	X =  247.902  mm,	Y =   -382.009  mm,	Z =   -256.245  mm,
	W =  90.000 deg,	P =   0.000 deg,	R =   90.000 deg
};
P[319]{
   GP1:
	UF : 0, UT : 6,		CONFIG : 'N U T, 0, 0, 0',
	X =  248.616  mm,	Y =   -381.594  mm,	Z =   -256.279  mm,
	W =  90.000 deg,	P =   0.000 deg,	R =   90.000 deg
};
P[320]{
   GP1:
	UF : 0, UT : 6,		CONFIG : 'N U T, 0, 0, 0',
	X =  254.561  mm,	Y =   -378.161  mm,	Z =   -256.286  mm,
	W =  90.000 deg,	P =   0.000 deg,	R =   90.000 deg
};
P[321]{
   GP1:
	UF : 0, UT : 6,		CONFIG : 'N U T, 0, 0, 0',
	X =  255.267  mm,	Y =   -377.759  mm,	Z =   -256.214  mm,
	W =  90.000 deg,	P =   0.000 deg,	R =   90.000 deg
};
P[322]{
   GP1:
	UF : 0, UT : 6,		CONFIG : 'N U T, 0, 0, 0',
	X =  258.215  mm,	Y =   -376.051  mm,	Z =   -256.285  mm,
	W =  90.000 deg,	P =   0.000 deg,	R =   90.000 deg
};
P[323]{
   GP1:
	UF : 0, UT : 6,		CONFIG : 'N U T, 0, 0, 0',
	X =  261.977  mm,	Y =   -373.884  mm,	Z =   -256.215  mm,
	W =  90.000 deg,	P =   0.000 deg,	R =   90.000 deg
};
P[324]{
   GP1:
	UF : 0, UT : 6,		CONFIG : 'N U T, 0, 0, 0',
	X =  262.661  mm,	Y =   -373.497  mm,	Z =   -256.123  mm,
	W =  90.000 deg,	P =   0.000 deg,	R =   90.000 deg
};
P[325]{
   GP1:
	UF : 0, UT : 6,		CONFIG : 'N U T, 0, 0, 0',
	X =  263.369  mm,	Y =   -373.079  mm,	Z =   -256.244  mm,
	W =  90.000 deg,	P =   0.000 deg,	R =   90.000 deg
};
P[326]{
   GP1:
	UF : 0, UT : 6,		CONFIG : 'N U T, 0, 0, 0',
	X =  265.622  mm,	Y =   -371.779  mm,	Z =   -256.224  mm,
	W =  90.000 deg,	P =   0.000 deg,	R =   90.000 deg
};
P[327]{
   GP1:
	UF : 0, UT : 6,		CONFIG : 'N U T, 0, 0, 0',
	X =  267.023  mm,	Y =   -370.977  mm,	Z =   -256.135  mm,
	W =  90.000 deg,	P =   0.000 deg,	R =   90.000 deg
};
P[328]{
   GP1:
	UF : 0, UT : 6,		CONFIG : 'N U T, 0, 0, 0',
	X =  267.777  mm,	Y =   -370.522  mm,	Z =   -256.283  mm,
	W =  90.000 deg,	P =   0.000 deg,	R =   90.000 deg
};
P[329]{
   GP1:
	UF : 0, UT : 6,		CONFIG : 'N U T, 0, 0, 0',
	X =  269.721  mm,	Y =   -369.001  mm,	Z =   -256.087  mm,
	W =  90.000 deg,	P =   0.000 deg,	R =   90.000 deg
};
P[330]{
   GP1:
	UF : 0, UT : 6,		CONFIG : 'N U T, 0, 0, 0',
	X =  269.875  mm,	Y =   -368.853  mm,	Z =   -255.819  mm,
	W =  90.000 deg,	P =   0.000 deg,	R =   90.000 deg
};
P[331]{
   GP1:
	UF : 0, UT : 6,		CONFIG : 'N U T, 0, 0, 0',
	X =  270.416  mm,	Y =   -368.129  mm,	Z =   -256.212  mm,
	W =  90.000 deg,	P =   0.000 deg,	R =   90.000 deg
};
P[332]{
   GP1:
	UF : 0, UT : 6,		CONFIG : 'N U T, 0, 0, 0',
	X =  270.805  mm,	Y =   -367.534  mm,	Z =   -256.111  mm,
	W =  90.000 deg,	P =   0.000 deg,	R =   90.000 deg
};
P[333]{
   GP1:
	UF : 0, UT : 6,		CONFIG : 'N U T, 0, 0, 0',
	X =  270.994  mm,	Y =   -367.194  mm,	Z =   -256.250  mm,
	W =  90.000 deg,	P =   0.000 deg,	R =   90.000 deg
};
P[334]{
   GP1:
	UF : 0, UT : 6,		CONFIG : 'N U T, 0, 0, 0',
	X =  271.729  mm,	Y =   -365.277  mm,	Z =   -256.239  mm,
	W =  90.000 deg,	P =   0.000 deg,	R =   90.000 deg
};
P[335]{
   GP1:
	UF : 0, UT : 6,		CONFIG : 'N U T, 0, 0, 0',
	X =  271.851  mm,	Y =   -361.616  mm,	Z =   -256.115  mm,
	W =  90.000 deg,	P =   0.000 deg,	R =   90.000 deg
};
P[336]{
   GP1:
	UF : 0, UT : 6,		CONFIG : 'N U T, 0, 0, 0',
	X =  271.727  mm,	Y =   -361.053  mm,	Z =   -256.193  mm,
	W =  90.000 deg,	P =   0.000 deg,	R =   90.000 deg
};
P[337]{
   GP1:
	UF : 0, UT : 6,		CONFIG : 'N U T, 0, 0, 0',
	X =  270.444  mm,	Y =   -358.219  mm,	Z =   -256.266  mm,
	W =  90.000 deg,	P =   0.000 deg,	R =   90.000 deg
};
P[338]{
   GP1:
	UF : 0, UT : 6,		CONFIG : 'N U T, 0, 0, 0',
	X =  270.041  mm,	Y =   -357.511  mm,	Z =   -256.196  mm,
	W =  90.000 deg,	P =   0.000 deg,	R =   90.000 deg
};
P[339]{
   GP1:
	UF : 0, UT : 6,		CONFIG : 'N U T, 0, 0, 0',
	X =  268.750  mm,	Y =   -355.278  mm,	Z =   -256.223  mm,
	W =  90.000 deg,	P =   0.000 deg,	R =   90.000 deg
};
P[340]{
   GP1:
	UF : 0, UT : 6,		CONFIG : 'N U T, 0, 0, 0',
	X =  267.926  mm,	Y =   -353.854  mm,	Z =   -256.236  mm,
	W =  90.000 deg,	P =   0.000 deg,	R =   90.000 deg
};
P[341]{
   GP1:
	UF : 0, UT : 6,		CONFIG : 'N U T, 0, 0, 0',
	X =  266.617  mm,	Y =   -351.583  mm,	Z =   -256.210  mm,
	W =  90.000 deg,	P =   0.000 deg,	R =   90.000 deg
};
P[342]{
   GP1:
	UF : 0, UT : 6,		CONFIG : 'N U T, 0, 0, 0',
	X =  265.790  mm,	Y =   -350.160  mm,	Z =   -256.269  mm,
	W =  90.000 deg,	P =   0.000 deg,	R =   90.000 deg
};
P[343]{
   GP1:
	UF : 0, UT : 6,		CONFIG : 'N U T, 0, 0, 0',
	X =  265.369  mm,	Y =   -349.416  mm,	Z =   -256.174  mm,
	W =  90.000 deg,	P =   0.000 deg,	R =   90.000 deg
};
P[344]{
   GP1:
	UF : 0, UT : 6,		CONFIG : 'N U T, 0, 0, 0',
	X =  264.933  mm,	Y =   -348.670  mm,	Z =   -256.231  mm,
	W =  90.000 deg,	P =   0.000 deg,	R =   90.000 deg
};
P[345]{
   GP1:
	UF : 0, UT : 6,		CONFIG : 'N U T, 0, 0, 0',
	X =  264.491  mm,	Y =   -347.910  mm,	Z =   -256.272  mm,
	W =  90.000 deg,	P =   0.000 deg,	R =   90.000 deg
};
P[346]{
   GP1:
	UF : 0, UT : 6,		CONFIG : 'N U T, 0, 0, 0',
	X =  264.090  mm,	Y =   -347.215  mm,	Z =   -256.262  mm,
	W =  90.000 deg,	P =   0.000 deg,	R =   90.000 deg
};
P[347]{
   GP1:
	UF : 0, UT : 6,		CONFIG : 'N U T, 0, 0, 0',
	X =  262.830  mm,	Y =   -345.031  mm,	Z =   -256.263  mm,
	W =  90.000 deg,	P =   0.000 deg,	R =   90.000 deg
};
P[348]{
   GP1:
	UF : 0, UT : 6,		CONFIG : 'N U T, 0, 0, 0',
	X =  262.368  mm,	Y =   -344.233  mm,	Z =   -256.279  mm,
	W =  90.000 deg,	P =   0.000 deg,	R =   90.000 deg
};
P[349]{
   GP1:
	UF : 0, UT : 6,		CONFIG : 'N U T, 0, 0, 0',
	X =  262.026  mm,	Y =   -343.628  mm,	Z =   -256.184  mm,
	W =  90.000 deg,	P =   0.000 deg,	R =   90.000 deg
};
P[350]{
   GP1:
	UF : 0, UT : 6,		CONFIG : 'N U T, 0, 0, 0',
	X =  260.236  mm,	Y =   -340.533  mm,	Z =   -256.219  mm,
	W =  90.000 deg,	P =   0.000 deg,	R =   90.000 deg
};
P[351]{
   GP1:
	UF : 0, UT : 6,		CONFIG : 'N U T, 0, 0, 0',
	X =  259.438  mm,	Y =   -339.161  mm,	Z =   -256.290  mm,
	W =  90.000 deg,	P =   0.000 deg,	R =   90.000 deg
};
P[352]{
   GP1:
	UF : 0, UT : 6,		CONFIG : 'N U T, 0, 0, 0',
	X =  258.110  mm,	Y =   -336.856  mm,	Z =   -256.255  mm,
	W =  90.000 deg,	P =   0.000 deg,	R =   90.000 deg
};
P[353]{
   GP1:
	UF : 0, UT : 6,		CONFIG : 'N U T, 0, 0, 0',
	X =  257.689  mm,	Y =   -336.131  mm,	Z =   -256.291  mm,
	W =  90.000 deg,	P =   0.000 deg,	R =   90.000 deg
};
P[354]{
   GP1:
	UF : 0, UT : 6,		CONFIG : 'N U T, 0, 0, 0',
	X =  256.431  mm,	Y =   -333.937  mm,	Z =   -256.170  mm,
	W =  90.000 deg,	P =   0.000 deg,	R =   90.000 deg
};
P[355]{
   GP1:
	UF : 0, UT : 6,		CONFIG : 'N U T, 0, 0, 0',
	X =  255.567  mm,	Y =   -332.445  mm,	Z =   -256.199  mm,
	W =  90.000 deg,	P =   0.000 deg,	R =   90.000 deg
};
P[356]{
   GP1:
	UF : 0, UT : 6,		CONFIG : 'N U T, 0, 0, 0',
	X =  255.156  mm,	Y =   -331.729  mm,	Z =   -256.181  mm,
	W =  90.000 deg,	P =   0.000 deg,	R =   90.000 deg
};
P[357]{
   GP1:
	UF : 0, UT : 6,		CONFIG : 'N U T, 0, 0, 0',
	X =  254.665  mm,	Y =   -330.894  mm,	Z =   -256.283  mm,
	W =  90.000 deg,	P =   0.000 deg,	R =   90.000 deg
};
P[358]{
   GP1:
	UF : 0, UT : 6,		CONFIG : 'N U T, 0, 0, 0',
	X =  254.295  mm,	Y =   -330.269  mm,	Z =   -256.272  mm,
	W =  90.000 deg,	P =   0.000 deg,	R =   90.000 deg
};
P[359]{
   GP1:
	UF : 0, UT : 6,		CONFIG : 'N U T, 0, 0, 0',
	X =  253.269  mm,	Y =   -328.882  mm,	Z =   -256.236  mm,
	W =  90.000 deg,	P =   0.000 deg,	R =   90.000 deg
};
P[360]{
   GP1:
	UF : 0, UT : 6,		CONFIG : 'N U T, 0, 0, 0',
	X =  252.851  mm,	Y =   -328.417  mm,	Z =   -256.192  mm,
	W =  90.000 deg,	P =   0.000 deg,	R =   90.000 deg
};
P[361]{
   GP1:
	UF : 0, UT : 6,		CONFIG : 'N U T, 0, 0, 0',
	X =  252.558  mm,	Y =   -328.182  mm,	Z =   -256.287  mm,
	W =  90.000 deg,	P =   0.000 deg,	R =   90.000 deg
};
P[362]{
   GP1:
	UF : 0, UT : 6,		CONFIG : 'N U T, 0, 0, 0',
	X =  251.892  mm,	Y =   -327.641  mm,	Z =   -256.229  mm,
	W =  90.000 deg,	P =   0.000 deg,	R =   90.000 deg
};
P[363]{
   GP1:
	UF : 0, UT : 6,		CONFIG : 'N U T, 0, 0, 0',
	X =  251.459  mm,	Y =   -327.358  mm,	Z =   -256.187  mm,
	W =  90.000 deg,	P =   0.000 deg,	R =   90.000 deg
};
P[364]{
   GP1:
	UF : 0, UT : 6,		CONFIG : 'N U T, 0, 0, 0',
	X =  249.222  mm,	Y =   -326.377  mm,	Z =   -256.167  mm,
	W =  90.000 deg,	P =   0.000 deg,	R =   90.000 deg
};
P[365]{
   GP1:
	UF : 0, UT : 6,		CONFIG : 'N U T, 0, 0, 0',
	X =  248.144  mm,	Y =   -326.165  mm,	Z =   -256.273  mm,
	W =  90.000 deg,	P =   0.000 deg,	R =   90.000 deg
};
P[366]{
   GP1:
	UF : 0, UT : 6,		CONFIG : 'N U T, 0, 0, 0',
	X =  247.391  mm,	Y =   -326.065  mm,	Z =   -256.154  mm,
	W =  90.000 deg,	P =   0.000 deg,	R =   90.000 deg
};
P[367]{
   GP1:
	UF : 0, UT : 6,		CONFIG : 'N U T, 0, 0, 0',
	X =  246.118  mm,	Y =   -326.120  mm,	Z =   -256.195  mm,
	W =  90.000 deg,	P =   0.000 deg,	R =   90.000 deg
};
P[368]{
   GP1:
	UF : 0, UT : 6,		CONFIG : 'N U T, 0, 0, 0',
	X =  244.973  mm,	Y =   -326.275  mm,	Z =   -255.877  mm,
	W =  90.000 deg,	P =   0.000 deg,	R =   90.000 deg
};
P[369]{
   GP1:
	UF : 0, UT : 6,		CONFIG : 'N U T, 0, 0, 0',
	X =  244.461  mm,	Y =   -326.465  mm,	Z =   -256.182  mm,
	W =  90.000 deg,	P =   0.000 deg,	R =   90.000 deg
};
P[370]{
   GP1:
	UF : 0, UT : 6,		CONFIG : 'N U T, 0, 0, 0',
	X =  242.026  mm,	Y =   -327.612  mm,	Z =   -256.201  mm,
	W =  90.000 deg,	P =   0.000 deg,	R =   90.000 deg
};
P[371]{
   GP1:
	UF : 0, UT : 6,		CONFIG : 'N U T, 0, 0, 0',
	X =  241.272  mm,	Y =   -328.043  mm,	Z =   -256.156  mm,
	W =  90.000 deg,	P =   0.000 deg,	R =   90.000 deg
};
P[372]{
   GP1:
	UF : 0, UT : 6,		CONFIG : 'N U T, 0, 0, 0',
	X =  240.597  mm,	Y =   -328.438  mm,	Z =   -256.220  mm,
	W =  90.000 deg,	P =   0.000 deg,	R =   90.000 deg
};
P[373]{
   GP1:
	UF : 0, UT : 6,		CONFIG : 'N U T, 0, 0, 0',
	X =  239.869  mm,	Y =   -328.863  mm,	Z =   -256.275  mm,
	W =  90.000 deg,	P =   0.000 deg,	R =   90.000 deg
};
P[374]{
   GP1:
	UF : 0, UT : 6,		CONFIG : 'N U T, 0, 0, 0',
	X =  239.046  mm,	Y =   -329.332  mm,	Z =   -256.198  mm,
	W =  90.000 deg,	P =   0.000 deg,	R =   90.000 deg
};
P[375]{
   GP1:
	UF : 0, UT : 6,		CONFIG : 'N U T, 0, 0, 0',
	X =  236.149  mm,	Y =   -331.005  mm,	Z =   -256.201  mm,
	W =  90.000 deg,	P =   0.000 deg,	R =   90.000 deg
};
P[376]{
   GP1:
	UF : 0, UT : 6,		CONFIG : 'N U T, 0, 0, 0',
	X =  234.723  mm,	Y =   -331.834  mm,	Z =   -256.270  mm,
	W =  90.000 deg,	P =   0.000 deg,	R =   90.000 deg
};
P[377]{
   GP1:
	UF : 0, UT : 6,		CONFIG : 'N U T, 0, 0, 0',
	X =  233.937  mm,	Y =   -332.289  mm,	Z =   -256.289  mm,
	W =  90.000 deg,	P =   0.000 deg,	R =   90.000 deg
};
P[378]{
   GP1:
	UF : 0, UT : 6,		CONFIG : 'N U T, 0, 0, 0',
	X =  233.257  mm,	Y =   -332.681  mm,	Z =   -256.279  mm,
	W =  90.000 deg,	P =   0.000 deg,	R =   90.000 deg
};
P[379]{
   GP1:
	UF : 0, UT : 6,		CONFIG : 'N U T, 0, 0, 0',
	X =  232.524  mm,	Y =   -333.105  mm,	Z =   -256.284  mm,
	W =  90.000 deg,	P =   0.000 deg,	R =   90.000 deg
};
P[380]{
   GP1:
	UF : 0, UT : 6,		CONFIG : 'N U T, 0, 0, 0',
	X =  231.761  mm,	Y =   -333.543  mm,	Z =   -256.260  mm,
	W =  90.000 deg,	P =   0.000 deg,	R =   90.000 deg
};
P[381]{
   GP1:
	UF : 0, UT : 6,		CONFIG : 'N U T, 0, 0, 0',
	X =  230.964  mm,	Y =   -333.998  mm,	Z =   -256.198  mm,
	W =  90.000 deg,	P =   0.000 deg,	R =   90.000 deg
};
P[382]{
   GP1:
	UF : 0, UT : 6,		CONFIG : 'N U T, 0, 0, 0',
	X =  230.308  mm,	Y =   -334.378  mm,	Z =   -256.209  mm,
	W =  90.000 deg,	P =   0.000 deg,	R =   90.000 deg
};
P[383]{
   GP1:
	UF : 0, UT : 6,		CONFIG : 'N U T, 0, 0, 0',
	X =  228.762  mm,	Y =   -335.273  mm,	Z =   -256.235  mm,
	W =  90.000 deg,	P =   0.000 deg,	R =   90.000 deg
};
P[384]{
   GP1:
	UF : 0, UT : 6,		CONFIG : 'N U T, 0, 0, 0',
	X =  226.535  mm,	Y =   -336.563  mm,	Z =   -256.285  mm,
	W =  90.000 deg,	P =   0.000 deg,	R =   90.000 deg
};
P[385]{
   GP1:
	UF : 0, UT : 6,		CONFIG : 'N U T, 0, 0, 0',
	X =  225.039  mm,	Y =   -337.426  mm,	Z =   -256.282  mm,
	W =  90.000 deg,	P =   0.000 deg,	R =   90.000 deg
};
P[386]{
   GP1:
	UF : 0, UT : 6,		CONFIG : 'N U T, 0, 0, 0',
	X =  224.460  mm,	Y =   -337.761  mm,	Z =   -256.294  mm,
	W =  90.000 deg,	P =   0.000 deg,	R =   90.000 deg
};
P[387]{
   GP1:
	UF : 0, UT : 6,		CONFIG : 'N U T, 0, 0, 0',
	X =  222.903  mm,	Y =   -338.653  mm,	Z =   -256.193  mm,
	W =  90.000 deg,	P =   0.000 deg,	R =   90.000 deg
};
P[388]{
   GP1:
	UF : 0, UT : 6,		CONFIG : 'N U T, 0, 0, 0',
	X =  218.417  mm,	Y =   -341.244  mm,	Z =   -256.213  mm,
	W =  90.000 deg,	P =   0.000 deg,	R =   90.000 deg
};
P[389]{
   GP1:
	UF : 0, UT : 6,		CONFIG : 'N U T, 0, 0, 0',
	X =  217.647  mm,	Y =   -341.694  mm,	Z =   -256.278  mm,
	W =  90.000 deg,	P =   0.000 deg,	R =   90.000 deg
};
P[390]{
   GP1:
	UF : 0, UT : 6,		CONFIG : 'N U T, 0, 0, 0',
	X =  214.021  mm,	Y =   -343.783  mm,	Z =   -256.220  mm,
	W =  90.000 deg,	P =   0.000 deg,	R =   90.000 deg
};
P[391]{
   GP1:
	UF : 0, UT : 6,		CONFIG : 'N U T, 0, 0, 0',
	X =  212.512  mm,	Y =   -344.659  mm,	Z =   -256.271  mm,
	W =  90.000 deg,	P =   0.000 deg,	R =   90.000 deg
};
P[392]{
   GP1:
	UF : 0, UT : 6,		CONFIG : 'N U T, 0, 0, 0',
	X =  211.156  mm,	Y =   -345.440  mm,	Z =   -256.255  mm,
	W =  90.000 deg,	P =   0.000 deg,	R =   90.000 deg
};
P[393]{
   GP1:
	UF : 0, UT : 6,		CONFIG : 'N U T, 0, 0, 0',
	X =  210.447  mm,	Y =   -345.848  mm,	Z =   -256.237  mm,
	W =  90.000 deg,	P =   0.000 deg,	R =   90.000 deg
};
P[394]{
   GP1:
	UF : 0, UT : 6,		CONFIG : 'N U T, 0, 0, 0',
	X =  208.242  mm,	Y =   -347.121  mm,	Z =   -256.243  mm,
	W =  90.000 deg,	P =   0.000 deg,	R =   90.000 deg
};
P[395]{
   GP1:
	UF : 0, UT : 6,		CONFIG : 'N U T, 0, 0, 0',
	X =  207.402  mm,	Y =   -347.608  mm,	Z =   -256.253  mm,
	W =  90.000 deg,	P =   0.000 deg,	R =   90.000 deg
};
P[396]{
   GP1:
	UF : 0, UT : 6,		CONFIG : 'N U T, 0, 0, 0',
	X =  205.941  mm,	Y =   -348.452  mm,	Z =   -256.265  mm,
	W =  90.000 deg,	P =   0.000 deg,	R =   90.000 deg
};
P[397]{
   GP1:
	UF : 0, UT : 6,		CONFIG : 'N U T, 0, 0, 0',
	X =  205.190  mm,	Y =   -348.882  mm,	Z =   -256.221  mm,
	W =  90.000 deg,	P =   0.000 deg,	R =   90.000 deg
};
P[398]{
   GP1:
	UF : 0, UT : 6,		CONFIG : 'N U T, 0, 0, 0',
	X =  202.336  mm,	Y =   -350.530  mm,	Z =   -256.224  mm,
	W =  90.000 deg,	P =   0.000 deg,	R =   90.000 deg
};
P[399]{
   GP1:
	UF : 0, UT : 6,		CONFIG : 'N U T, 0, 0, 0',
	X =  200.125  mm,	Y =   -351.810  mm,	Z =   -256.270  mm,
	W =  90.000 deg,	P =   0.000 deg,	R =   90.000 deg
};
P[400]{
   GP1:
	UF : 0, UT : 6,		CONFIG : 'N U T, 0, 0, 0',
	X =  198.501  mm,	Y =   -352.750  mm,	Z =   -256.289  mm,
	W =  90.000 deg,	P =   0.000 deg,	R =   90.000 deg
};
P[401]{
   GP1:
	UF : 0, UT : 6,		CONFIG : 'N U T, 0, 0, 0',
	X =  197.783  mm,	Y =   -353.163  mm,	Z =   -256.274  mm,
	W =  90.000 deg,	P =   0.000 deg,	R =   90.000 deg
};
P[402]{
   GP1:
	UF : 0, UT : 6,		CONFIG : 'N U T, 0, 0, 0',
	X =  196.032  mm,	Y =   -353.414  mm,	Z =   -246.859  mm,
	W =  90.000 deg,	P =   0.000 deg,	R =   90.000 deg
};
P[403]{
   GP1:
	UF : 0, UT : 6,		CONFIG : 'N U T, 0, 0, 0',
	X =  195.473  mm,	Y =   -353.741  mm,	Z =   -246.915  mm,
	W =  90.000 deg,	P =   0.000 deg,	R =   90.000 deg
};
P[404]{
   GP1:
	UF : 0, UT : 6,		CONFIG : 'N U T, 0, 0, 0',
	X =  194.619  mm,	Y =   -354.233  mm,	Z =   -246.902  mm,
	W =  90.000 deg,	P =   0.000 deg,	R =   90.000 deg
};
P[405]{
   GP1:
	UF : 0, UT : 6,		CONFIG : 'N U T, 0, 0, 0',
	X =  193.731  mm,	Y =   -354.745  mm,	Z =   -246.888  mm,
	W =  90.000 deg,	P =   0.000 deg,	R =   90.000 deg
};
P[406]{
   GP1:
	UF : 0, UT : 6,		CONFIG : 'N U T, 0, 0, 0',
	X =  193.023  mm,	Y =   -355.154  mm,	Z =   -246.887  mm,
	W =  90.000 deg,	P =   0.000 deg,	R =   90.000 deg
};
P[407]{
   GP1:
	UF : 0, UT : 6,		CONFIG : 'N U T, 0, 0, 0',
	X =  192.356  mm,	Y =   -355.536  mm,	Z =   -246.860  mm,
	W =  90.000 deg,	P =   0.000 deg,	R =   90.000 deg
};
P[408]{
   GP1:
	UF : 0, UT : 6,		CONFIG : 'N U T, 0, 0, 0',
	X =  190.808  mm,	Y =   -356.432  mm,	Z =   -246.883  mm,
	W =  90.000 deg,	P =   0.000 deg,	R =   90.000 deg
};
P[409]{
   GP1:
	UF : 0, UT : 6,		CONFIG : 'N U T, 0, 0, 0',
	X =  190.217  mm,	Y =   -356.774  mm,	Z =   -246.892  mm,
	W =  90.000 deg,	P =   0.000 deg,	R =   90.000 deg
};
P[410]{
   GP1:
	UF : 0, UT : 6,		CONFIG : 'N U T, 0, 0, 0',
	X =  189.373  mm,	Y =   -357.263  mm,	Z =   -246.919  mm,
	W =  90.000 deg,	P =   0.000 deg,	R =   90.000 deg
};
P[411]{
   GP1:
	UF : 0, UT : 6,		CONFIG : 'N U T, 0, 0, 0',
	X =  188.668  mm,	Y =   -357.657  mm,	Z =   -246.758  mm,
	W =  90.000 deg,	P =   0.000 deg,	R =   90.000 deg
};
P[412]{
   GP1:
	UF : 0, UT : 6,		CONFIG : 'N U T, 0, 0, 0',
	X =  188.044  mm,	Y =   -358.028  mm,	Z =   -246.877  mm,
	W =  90.000 deg,	P =   0.000 deg,	R =   90.000 deg
};
P[413]{
   GP1:
	UF : 0, UT : 6,		CONFIG : 'N U T, 0, 0, 0',
	X =  187.147  mm,	Y =   -358.547  mm,	Z =   -246.893  mm,
	W =  90.000 deg,	P =   0.000 deg,	R =   90.000 deg
};
P[414]{
   GP1:
	UF : 0, UT : 6,		CONFIG : 'N U T, 0, 0, 0',
	X =  186.476  mm,	Y =   -358.932  mm,	Z =   -246.874  mm,
	W =  90.000 deg,	P =   0.000 deg,	R =   90.000 deg
};
P[415]{
   GP1:
	UF : 0, UT : 6,		CONFIG : 'N U T, 0, 0, 0',
	X =  185.037  mm,	Y =   -359.767  mm,	Z =   -246.923  mm,
	W =  90.000 deg,	P =   0.000 deg,	R =   90.000 deg
};
P[416]{
   GP1:
	UF : 0, UT : 6,		CONFIG : 'N U T, 0, 0, 0',
	X =  183.547  mm,	Y =   -360.627  mm,	Z =   -246.906  mm,
	W =  90.000 deg,	P =   0.000 deg,	R =   90.000 deg
};
P[417]{
   GP1:
	UF : 0, UT : 6,		CONFIG : 'N U T, 0, 0, 0',
	X =  182.141  mm,	Y =   -361.440  mm,	Z =   -246.921  mm,
	W =  90.000 deg,	P =   0.000 deg,	R =   90.000 deg
};
P[418]{
   GP1:
	UF : 0, UT : 6,		CONFIG : 'N U T, 0, 0, 0',
	X =  180.536  mm,	Y =   -362.357  mm,	Z =   -246.812  mm,
	W =  90.000 deg,	P =   0.000 deg,	R =   90.000 deg
};
P[419]{
   GP1:
	UF : 0, UT : 6,		CONFIG : 'N U T, 0, 0, 0',
	X =  178.442  mm,	Y =   -363.573  mm,	Z =   -246.894  mm,
	W =  90.000 deg,	P =   0.000 deg,	R =   90.000 deg
};
P[420]{
   GP1:
	UF : 0, UT : 6,		CONFIG : 'N U T, 0, 0, 0',
	X =  175.338  mm,	Y =   -365.357  mm,	Z =   -246.788  mm,
	W =  90.000 deg,	P =   0.000 deg,	R =   90.000 deg
};
P[421]{
   GP1:
	UF : 0, UT : 6,		CONFIG : 'N U T, 0, 0, 0',
	X =  174.572  mm,	Y =   -365.805  mm,	Z =   -246.864  mm,
	W =  90.000 deg,	P =   0.000 deg,	R =   90.000 deg
};
P[422]{
   GP1:
	UF : 0, UT : 6,		CONFIG : 'N U T, 0, 0, 0',
	X =  173.813  mm,	Y =   -366.240  mm,	Z =   -246.828  mm,
	W =  90.000 deg,	P =   0.000 deg,	R =   90.000 deg
};
P[423]{
   GP1:
	UF : 0, UT : 6,		CONFIG : 'N U T, 0, 0, 0',
	X =  173.280  mm,	Y =   -366.554  mm,	Z =   -246.906  mm,
	W =  90.000 deg,	P =   0.000 deg,	R =   90.000 deg
};
P[424]{
   GP1:
	UF : 0, UT : 6,		CONFIG : 'N U T, 0, 0, 0',
	X =  172.494  mm,	Y =   -367.005  mm,	Z =   -246.867  mm,
	W =  90.000 deg,	P =   0.000 deg,	R =   90.000 deg
};
P[425]{
   GP1:
	UF : 0, UT : 6,		CONFIG : 'N U T, 0, 0, 0',
	X =  171.741  mm,	Y =   -367.438  mm,	Z =   -246.840  mm,
	W =  90.000 deg,	P =   0.000 deg,	R =   90.000 deg
};
P[426]{
   GP1:
	UF : 0, UT : 6,		CONFIG : 'N U T, 0, 0, 0',
	X =  165.137  mm,	Y =   -371.244  mm,	Z =   -246.757  mm,
	W =  90.000 deg,	P =   0.000 deg,	R =   90.000 deg
};
P[427]{
   GP1:
	UF : 0, UT : 6,		CONFIG : 'N U T, 0, 0, 0',
	X =  164.370  mm,	Y =   -371.694  mm,	Z =   -246.846  mm,
	W =  90.000 deg,	P =   0.000 deg,	R =   90.000 deg
};
P[428]{
   GP1:
	UF : 0, UT : 6,		CONFIG : 'N U T, 0, 0, 0',
	X =  162.155  mm,	Y =   -372.976  mm,	Z =   -246.883  mm,
	W =  90.000 deg,	P =   0.000 deg,	R =   90.000 deg
};
P[429]{
   GP1:
	UF : 0, UT : 6,		CONFIG : 'N U T, 0, 0, 0',
	X =  161.482  mm,	Y =   -373.364  mm,	Z =   -246.882  mm,
	W =  90.000 deg,	P =   0.000 deg,	R =   90.000 deg
};
P[430]{
   GP1:
	UF : 0, UT : 6,		CONFIG : 'N U T, 0, 0, 0',
	X =  159.173  mm,	Y =   -374.702  mm,	Z =   -246.936  mm,
	W =  90.000 deg,	P =   0.000 deg,	R =   90.000 deg
};
P[431]{
   GP1:
	UF : 0, UT : 6,		CONFIG : 'N U T, 0, 0, 0',
	X =  157.850  mm,	Y =   -375.464  mm,	Z =   -246.904  mm,
	W =  90.000 deg,	P =   0.000 deg,	R =   90.000 deg
};
P[432]{
   GP1:
	UF : 0, UT : 6,		CONFIG : 'N U T, 0, 0, 0',
	X =  157.104  mm,	Y =   -375.894  mm,	Z =   -246.913  mm,
	W =  90.000 deg,	P =   0.000 deg,	R =   90.000 deg
};
P[433]{
   GP1:
	UF : 0, UT : 6,		CONFIG : 'N U T, 0, 0, 0',
	X =  156.303  mm,	Y =   -376.357  mm,	Z =   -246.902  mm,
	W =  90.000 deg,	P =   0.000 deg,	R =   90.000 deg
};
P[434]{
   GP1:
	UF : 0, UT : 6,		CONFIG : 'N U T, 0, 0, 0',
	X =  155.575  mm,	Y =   -376.775  mm,	Z =   -246.882  mm,
	W =  90.000 deg,	P =   0.000 deg,	R =   90.000 deg
};
P[435]{
   GP1:
	UF : 0, UT : 6,		CONFIG : 'N U T, 0, 0, 0',
	X =  154.766  mm,	Y =   -377.245  mm,	Z =   -246.920  mm,
	W =  90.000 deg,	P =   0.000 deg,	R =   90.000 deg
};
P[436]{
   GP1:
	UF : 0, UT : 6,		CONFIG : 'N U T, 0, 0, 0',
	X =  153.304  mm,	Y =   -378.087  mm,	Z =   -246.895  mm,
	W =  90.000 deg,	P =   0.000 deg,	R =   90.000 deg
};
P[437]{
   GP1:
	UF : 0, UT : 6,		CONFIG : 'N U T, 0, 0, 0',
	X =  151.755  mm,	Y =   -378.973  mm,	Z =   -246.785  mm,
	W =  90.000 deg,	P =   0.000 deg,	R =   90.000 deg
};
P[438]{
   GP1:
	UF : 0, UT : 6,		CONFIG : 'N U T, 0, 0, 0',
	X =  150.364  mm,	Y =   -379.899  mm,	Z =   -246.888  mm,
	W =  90.000 deg,	P =   0.000 deg,	R =   90.000 deg
};
P[439]{
   GP1:
	UF : 0, UT : 6,		CONFIG : 'N U T, 0, 0, 0',
	X =  150.052  mm,	Y =   -380.157  mm,	Z =   -246.874  mm,
	W =  90.000 deg,	P =   0.000 deg,	R =   90.000 deg
};
P[440]{
   GP1:
	UF : 0, UT : 6,		CONFIG : 'N U T, 0, 0, 0',
	X =  149.745  mm,	Y =   -380.438  mm,	Z =   -246.891  mm,
	W =  90.000 deg,	P =   0.000 deg,	R =   90.000 deg
};
P[441]{
   GP1:
	UF : 0, UT : 6,		CONFIG : 'N U T, 0, 0, 0',
	X =  148.142  mm,	Y =   -382.521  mm,	Z =   -246.875  mm,
	W =  90.000 deg,	P =   0.000 deg,	R =   90.000 deg
};
P[442]{
   GP1:
	UF : 0, UT : 6,		CONFIG : 'N U T, 0, 0, 0',
	X =  147.771  mm,	Y =   -383.319  mm,	Z =   -246.930  mm,
	W =  90.000 deg,	P =   0.000 deg,	R =   90.000 deg
};
P[443]{
   GP1:
	UF : 0, UT : 6,		CONFIG : 'N U T, 0, 0, 0',
	X =  147.532  mm,	Y =   -383.857  mm,	Z =   -246.754  mm,
	W =  90.000 deg,	P =   0.000 deg,	R =   90.000 deg
};
P[444]{
   GP1:
	UF : 0, UT : 6,		CONFIG : 'N U T, 0, 0, 0',
	X =  147.402  mm,	Y =   -384.384  mm,	Z =   -246.864  mm,
	W =  90.000 deg,	P =   0.000 deg,	R =   90.000 deg
};
P[445]{
   GP1:
	UF : 0, UT : 6,		CONFIG : 'N U T, 0, 0, 0',
	X =  147.134  mm,	Y =   -385.696  mm,	Z =   -246.600  mm,
	W =  90.000 deg,	P =   0.000 deg,	R =   90.000 deg
};
P[446]{
   GP1:
	UF : 0, UT : 6,		CONFIG : 'N U T, 0, 0, 0',
	X =  147.279  mm,	Y =   -388.188  mm,	Z =   -246.943  mm,
	W =  90.000 deg,	P =   0.000 deg,	R =   90.000 deg
};
P[447]{
   GP1:
	UF : 0, UT : 6,		CONFIG : 'N U T, 0, 0, 0',
	X =  148.149  mm,	Y =   -390.622  mm,	Z =   -246.907  mm,
	W =  90.000 deg,	P =   0.000 deg,	R =   90.000 deg
};
P[448]{
   GP1:
	UF : 0, UT : 6,		CONFIG : 'N U T, 0, 0, 0',
	X =  148.497  mm,	Y =   -391.271  mm,	Z =   -246.790  mm,
	W =  90.000 deg,	P =   0.000 deg,	R =   90.000 deg
};
P[449]{
   GP1:
	UF : 0, UT : 6,		CONFIG : 'N U T, 0, 0, 0',
	X =  148.965  mm,	Y =   -392.072  mm,	Z =   -246.867  mm,
	W =  90.000 deg,	P =   0.000 deg,	R =   90.000 deg
};
P[450]{
   GP1:
	UF : 0, UT : 6,		CONFIG : 'N U T, 0, 0, 0',
	X =  149.414  mm,	Y =   -392.844  mm,	Z =   -246.910  mm,
	W =  90.000 deg,	P =   0.000 deg,	R =   90.000 deg
};
P[451]{
   GP1:
	UF : 0, UT : 6,		CONFIG : 'N U T, 0, 0, 0',
	X =  149.794  mm,	Y =   -393.520  mm,	Z =   -246.782  mm,
	W =  90.000 deg,	P =   0.000 deg,	R =   90.000 deg
};
P[452]{
   GP1:
	UF : 0, UT : 6,		CONFIG : 'N U T, 0, 0, 0',
	X =  150.651  mm,	Y =   -394.989  mm,	Z =   -246.889  mm,
	W =  90.000 deg,	P =   0.000 deg,	R =   90.000 deg
};
P[453]{
   GP1:
	UF : 0, UT : 6,		CONFIG : 'N U T, 0, 0, 0',
	X =  151.967  mm,	Y =   -397.263  mm,	Z =   -246.922  mm,
	W =  90.000 deg,	P =   0.000 deg,	R =   90.000 deg
};
P[454]{
   GP1:
	UF : 0, UT : 6,		CONFIG : 'N U T, 0, 0, 0',
	X =  152.788  mm,	Y =   -398.684  mm,	Z =   -246.932  mm,
	W =  90.000 deg,	P =   0.000 deg,	R =   90.000 deg
};
P[455]{
   GP1:
	UF : 0, UT : 6,		CONFIG : 'N U T, 0, 0, 0',
	X =  153.223  mm,	Y =   -399.439  mm,	Z =   -246.919  mm,
	W =  90.000 deg,	P =   0.000 deg,	R =   90.000 deg
};
P[456]{
   GP1:
	UF : 0, UT : 6,		CONFIG : 'N U T, 0, 0, 0',
	X =  154.047  mm,	Y =   -400.880  mm,	Z =   -246.817  mm,
	W =  90.000 deg,	P =   0.000 deg,	R =   90.000 deg
};
P[457]{
   GP1:
	UF : 0, UT : 6,		CONFIG : 'N U T, 0, 0, 0',
	X =  154.441  mm,	Y =   -401.547  mm,	Z =   -246.933  mm,
	W =  90.000 deg,	P =   0.000 deg,	R =   90.000 deg
};
P[458]{
   GP1:
	UF : 0, UT : 6,		CONFIG : 'N U T, 0, 0, 0',
	X =  154.900  mm,	Y =   -402.355  mm,	Z =   -246.835  mm,
	W =  90.000 deg,	P =   0.000 deg,	R =   90.000 deg
};
P[459]{
   GP1:
	UF : 0, UT : 6,		CONFIG : 'N U T, 0, 0, 0',
	X =  156.137  mm,	Y =   -404.483  mm,	Z =   -246.939  mm,
	W =  90.000 deg,	P =   0.000 deg,	R =   90.000 deg
};
P[460]{
   GP1:
	UF : 0, UT : 6,		CONFIG : 'N U T, 0, 0, 0',
	X =  157.074  mm,	Y =   -406.107  mm,	Z =   -246.937  mm,
	W =  90.000 deg,	P =   0.000 deg,	R =   90.000 deg
};
P[461]{
   GP1:
	UF : 0, UT : 6,		CONFIG : 'N U T, 0, 0, 0',
	X =  157.463  mm,	Y =   -406.806  mm,	Z =   -246.751  mm,
	W =  90.000 deg,	P =   0.000 deg,	R =   90.000 deg
};
P[462]{
   GP1:
	UF : 0, UT : 6,		CONFIG : 'N U T, 0, 0, 0',
	X =  158.780  mm,	Y =   -409.069  mm,	Z =   -246.872  mm,
	W =  90.000 deg,	P =   0.000 deg,	R =   90.000 deg
};
P[463]{
   GP1:
	UF : 0, UT : 6,		CONFIG : 'N U T, 0, 0, 0',
	X =  160.417  mm,	Y =   -411.908  mm,	Z =   -246.847  mm,
	W =  90.000 deg,	P =   0.000 deg,	R =   90.000 deg
};
P[464]{
   GP1:
	UF : 0, UT : 6,		CONFIG : 'N U T, 0, 0, 0',
	X =  160.852  mm,	Y =   -412.665  mm,	Z =   -246.824  mm,
	W =  90.000 deg,	P =   0.000 deg,	R =   90.000 deg
};
P[465]{
   GP1:
	UF : 0, UT : 6,		CONFIG : 'N U T, 0, 0, 0',
	X =  162.182  mm,	Y =   -414.959  mm,	Z =   -246.889  mm,
	W =  90.000 deg,	P =   0.000 deg,	R =   90.000 deg
};
P[466]{
   GP1:
	UF : 0, UT : 6,		CONFIG : 'N U T, 0, 0, 0',
	X =  162.993  mm,	Y =   -416.369  mm,	Z =   -246.854  mm,
	W =  90.000 deg,	P =   0.000 deg,	R =   90.000 deg
};
P[467]{
   GP1:
	UF : 0, UT : 6,		CONFIG : 'N U T, 0, 0, 0',
	X =  163.433  mm,	Y =   -417.133  mm,	Z =   -246.838  mm,
	W =  90.000 deg,	P =   0.000 deg,	R =   90.000 deg
};
P[468]{
   GP1:
	UF : 0, UT : 6,		CONFIG : 'N U T, 0, 0, 0',
	X =  164.696  mm,	Y =   -419.325  mm,	Z =   -246.809  mm,
	W =  90.000 deg,	P =   0.000 deg,	R =   90.000 deg
};
P[469]{
   GP1:
	UF : 0, UT : 6,		CONFIG : 'N U T, 0, 0, 0',
	X =  165.120  mm,	Y =   -420.046  mm,	Z =   -246.901  mm,
	W =  90.000 deg,	P =   0.000 deg,	R =   90.000 deg
};
P[470]{
   GP1:
	UF : 0, UT : 6,		CONFIG : 'N U T, 0, 0, 0',
	X =  166.001  mm,	Y =   -421.426  mm,	Z =   -246.911  mm,
	W =  90.000 deg,	P =   0.000 deg,	R =   90.000 deg
};
P[471]{
   GP1:
	UF : 0, UT : 6,		CONFIG : 'N U T, 0, 0, 0',
	X =  166.363  mm,	Y =   -421.896  mm,	Z =   -246.672  mm,
	W =  90.000 deg,	P =   0.000 deg,	R =   90.000 deg
};
P[472]{
   GP1:
	UF : 0, UT : 6,		CONFIG : 'N U T, 0, 0, 0',
	X =  166.597  mm,	Y =   -422.122  mm,	Z =   -246.919  mm,
	W =  90.000 deg,	P =   0.000 deg,	R =   90.000 deg
};
P[473]{
   GP1:
	UF : 0, UT : 6,		CONFIG : 'N U T, 0, 0, 0',
	X =  167.939  mm,	Y =   -423.294  mm,	Z =   -246.879  mm,
	W =  90.000 deg,	P =   0.000 deg,	R =   90.000 deg
};
P[474]{
   GP1:
	UF : 0, UT : 6,		CONFIG : 'N U T, 0, 0, 0',
	X =  169.552  mm,	Y =   -424.179  mm,	Z =   -246.826  mm,
	W =  90.000 deg,	P =   0.000 deg,	R =   90.000 deg
};
P[475]{
   GP1:
	UF : 0, UT : 6,		CONFIG : 'N U T, 0, 0, 0',
	X =  171.211  mm,	Y =   -424.676  mm,	Z =   -246.867  mm,
	W =  90.000 deg,	P =   0.000 deg,	R =   90.000 deg
};
P[476]{
   GP1:
	UF : 0, UT : 6,		CONFIG : 'N U T, 0, 0, 0',
	X =  173.500  mm,	Y =   -424.781  mm,	Z =   -246.935  mm,
	W =  90.000 deg,	P =   0.000 deg,	R =   90.000 deg
};
P[477]{
   GP1:
	UF : 0, UT : 6,		CONFIG : 'N U T, 0, 0, 0',
	X =  176.029  mm,	Y =   -424.176  mm,	Z =   -246.716  mm,
	W =  90.000 deg,	P =   0.000 deg,	R =   90.000 deg
};
P[478]{
   GP1:
	UF : 0, UT : 6,		CONFIG : 'N U T, 0, 0, 0',
	X =  178.937  mm,	Y =   -422.587  mm,	Z =   -246.855  mm,
	W =  90.000 deg,	P =   0.000 deg,	R =   90.000 deg
};
P[479]{
   GP1:
	UF : 0, UT : 6,		CONFIG : 'N U T, 0, 0, 0',
	X =  179.778  mm,	Y =   -422.096  mm,	Z =   -246.920  mm,
	W =  90.000 deg,	P =   0.000 deg,	R =   90.000 deg
};
P[480]{
   GP1:
	UF : 0, UT : 6,		CONFIG : 'N U T, 0, 0, 0',
	X =  181.226  mm,	Y =   -421.277  mm,	Z =   -246.711  mm,
	W =  90.000 deg,	P =   0.000 deg,	R =   90.000 deg
};
P[481]{
   GP1:
	UF : 0, UT : 6,		CONFIG : 'N U T, 0, 0, 0',
	X =  182.017  mm,	Y =   -420.803  mm,	Z =   -246.926  mm,
	W =  90.000 deg,	P =   0.000 deg,	R =   90.000 deg
};
P[482]{
   GP1:
	UF : 0, UT : 6,		CONFIG : 'N U T, 0, 0, 0',
	X =  182.721  mm,	Y =   -420.397  mm,	Z =   -246.912  mm,
	W =  90.000 deg,	P =   0.000 deg,	R =   90.000 deg
};
P[483]{
   GP1:
	UF : 0, UT : 6,		CONFIG : 'N U T, 0, 0, 0',
	X =  184.857  mm,	Y =   -419.169  mm,	Z =   -246.851  mm,
	W =  90.000 deg,	P =   0.000 deg,	R =   90.000 deg
};
P[484]{
   GP1:
	UF : 0, UT : 6,		CONFIG : 'N U T, 0, 0, 0',
	X =  186.319  mm,	Y =   -418.322  mm,	Z =   -246.886  mm,
	W =  90.000 deg,	P =   0.000 deg,	R =   90.000 deg
};
P[485]{
   GP1:
	UF : 0, UT : 6,		CONFIG : 'N U T, 0, 0, 0',
	X =  188.613  mm,	Y =   -417.003  mm,	Z =   -246.821  mm,
	W =  90.000 deg,	P =   0.000 deg,	R =   90.000 deg
};
P[486]{
   GP1:
	UF : 0, UT : 6,		CONFIG : 'N U T, 0, 0, 0',
	X =  189.289  mm,	Y =   -416.604  mm,	Z =   -246.930  mm,
	W =  90.000 deg,	P =   0.000 deg,	R =   90.000 deg
};
P[487]{
   GP1:
	UF : 0, UT : 6,		CONFIG : 'N U T, 0, 0, 0',
	X =  190.044  mm,	Y =   -416.171  mm,	Z =   -246.890  mm,
	W =  90.000 deg,	P =   0.000 deg,	R =   90.000 deg
};
P[488]{
   GP1:
	UF : 0, UT : 6,		CONFIG : 'N U T, 0, 0, 0',
	X =  191.502  mm,	Y =   -415.326  mm,	Z =   -246.923  mm,
	W =  90.000 deg,	P =   0.000 deg,	R =   90.000 deg
};
P[489]{
   GP1:
	UF : 0, UT : 6,		CONFIG : 'N U T, 0, 0, 0',
	X =  193.020  mm,	Y =   -414.456  mm,	Z =   -246.852  mm,
	W =  90.000 deg,	P =   0.000 deg,	R =   90.000 deg
};
P[490]{
   GP1:
	UF : 0, UT : 6,		CONFIG : 'N U T, 0, 0, 0',
	X =  193.810  mm,	Y =   -413.995  mm,	Z =   -246.906  mm,
	W =  90.000 deg,	P =   0.000 deg,	R =   90.000 deg
};
P[491]{
   GP1:
	UF : 0, UT : 6,		CONFIG : 'N U T, 0, 0, 0',
	X =  194.641  mm,	Y =   -413.515  mm,	Z =   -246.918  mm,
	W =  90.000 deg,	P =   0.000 deg,	R =   90.000 deg
};
P[492]{
   GP1:
	UF : 0, UT : 6,		CONFIG : 'N U T, 0, 0, 0',
	X =  195.229  mm,	Y =   -413.186  mm,	Z =   -246.785  mm,
	W =  90.000 deg,	P =   0.000 deg,	R =   90.000 deg
};
P[493]{
   GP1:
	UF : 0, UT : 6,		CONFIG : 'N U T, 0, 0, 0',
	X =  195.953  mm,	Y =   -412.757  mm,	Z =   -246.919  mm,
	W =  90.000 deg,	P =   0.000 deg,	R =   90.000 deg
};
P[494]{
   GP1:
	UF : 0, UT : 6,		CONFIG : 'N U T, 0, 0, 0',
	X =  198.249  mm,	Y =   -411.438  mm,	Z =   -246.827  mm,
	W =  90.000 deg,	P =   0.000 deg,	R =   90.000 deg
};
P[495]{
   GP1:
	UF : 0, UT : 6,		CONFIG : 'N U T, 0, 0, 0',
	X =  199.640  mm,	Y =   -410.628  mm,	Z =   -246.922  mm,
	W =  90.000 deg,	P =   0.000 deg,	R =   90.000 deg
};
P[496]{
   GP1:
	UF : 0, UT : 6,		CONFIG : 'N U T, 0, 0, 0',
	X =  200.391  mm,	Y =   -410.194  mm,	Z =   -246.923  mm,
	W =  90.000 deg,	P =   0.000 deg,	R =   90.000 deg
};
P[497]{
   GP1:
	UF : 0, UT : 6,		CONFIG : 'N U T, 0, 0, 0',
	X =  201.752  mm,	Y =   -409.411  mm,	Z =   -246.885  mm,
	W =  90.000 deg,	P =   0.000 deg,	R =   90.000 deg
};
P[498]{
   GP1:
	UF : 0, UT : 6,		CONFIG : 'N U T, 0, 0, 0',
	X =  204.104  mm,	Y =   -408.049  mm,	Z =   -246.943  mm,
	W =  90.000 deg,	P =   0.000 deg,	R =   90.000 deg
};
P[499]{
   GP1:
	UF : 0, UT : 6,		CONFIG : 'N U T, 0, 0, 0',
	X =  205.641  mm,	Y =   -407.163  mm,	Z =   -246.928  mm,
	W =  90.000 deg,	P =   0.000 deg,	R =   90.000 deg
};
P[500]{
   GP1:
	UF : 0, UT : 6,		CONFIG : 'N U T, 0, 0, 0',
	X =  206.214  mm,	Y =   -406.833  mm,	Z =   -246.911  mm,
	W =  90.000 deg,	P =   0.000 deg,	R =   90.000 deg
};
P[501]{
   GP1:
	UF : 0, UT : 6,		CONFIG : 'N U T, 0, 0, 0',
	X =  209.353  mm,	Y =   -405.022  mm,	Z =   -246.899  mm,
	W =  90.000 deg,	P =   0.000 deg,	R =   90.000 deg
};
P[502]{
   GP1:
	UF : 0, UT : 6,		CONFIG : 'N U T, 0, 0, 0',
	X =  212.277  mm,	Y =   -403.335  mm,	Z =   -246.877  mm,
	W =  90.000 deg,	P =   0.000 deg,	R =   90.000 deg
};
P[503]{
   GP1:
	UF : 0, UT : 6,		CONFIG : 'N U T, 0, 0, 0',
	X =  213.646  mm,	Y =   -402.542  mm,	Z =   -246.911  mm,
	W =  90.000 deg,	P =   0.000 deg,	R =   90.000 deg
};
P[504]{
   GP1:
	UF : 0, UT : 6,		CONFIG : 'N U T, 0, 0, 0',
	X =  214.373  mm,	Y =   -402.126  mm,	Z =   -246.862  mm,
	W =  90.000 deg,	P =   0.000 deg,	R =   90.000 deg
};
P[505]{
   GP1:
	UF : 0, UT : 6,		CONFIG : 'N U T, 0, 0, 0',
	X =  215.870  mm,	Y =   -401.256  mm,	Z =   -246.930  mm,
	W =  90.000 deg,	P =   0.000 deg,	R =   90.000 deg
};
P[506]{
   GP1:
	UF : 0, UT : 6,		CONFIG : 'N U T, 0, 0, 0',
	X =  216.623  mm,	Y =   -400.832  mm,	Z =   -246.796  mm,
	W =  90.000 deg,	P =   0.000 deg,	R =   90.000 deg
};
P[507]{
   GP1:
	UF : 0, UT : 6,		CONFIG : 'N U T, 0, 0, 0',
	X =  217.358  mm,	Y =   -400.397  mm,	Z =   -246.929  mm,
	W =  90.000 deg,	P =   0.000 deg,	R =   90.000 deg
};
P[508]{
   GP1:
	UF : 0, UT : 6,		CONFIG : 'N U T, 0, 0, 0',
	X =  220.260  mm,	Y =   -398.720  mm,	Z =   -246.942  mm,
	W =  90.000 deg,	P =   0.000 deg,	R =   90.000 deg
};
P[509]{
   GP1:
	UF : 0, UT : 6,		CONFIG : 'N U T, 0, 0, 0',
	X =  220.932  mm,	Y =   -398.341  mm,	Z =   -246.826  mm,
	W =  90.000 deg,	P =   0.000 deg,	R =   90.000 deg
};
P[510]{
   GP1:
	UF : 0, UT : 6,		CONFIG : 'N U T, 0, 0, 0',
	X =  221.803  mm,	Y =   -397.836  mm,	Z =   -246.869  mm,
	W =  90.000 deg,	P =   0.000 deg,	R =   90.000 deg
};
P[511]{
   GP1:
	UF : 0, UT : 6,		CONFIG : 'N U T, 0, 0, 0',
	X =  223.911  mm,	Y =   -396.616  mm,	Z =   -246.897  mm,
	W =  90.000 deg,	P =   0.000 deg,	R =   90.000 deg
};
P[512]{
   GP1:
	UF : 0, UT : 6,		CONFIG : 'N U T, 0, 0, 0',
	X =  225.367  mm,	Y =   -395.773  mm,	Z =   -246.925  mm,
	W =  90.000 deg,	P =   0.000 deg,	R =   90.000 deg
};
P[513]{
   GP1:
	UF : 0, UT : 6,		CONFIG : 'N U T, 0, 0, 0',
	X =  228.415  mm,	Y =   -394.021  mm,	Z =   -246.828  mm,
	W =  90.000 deg,	P =   0.000 deg,	R =   90.000 deg
};
P[514]{
   GP1:
	UF : 0, UT : 6,		CONFIG : 'N U T, 0, 0, 0',
	X =  230.540  mm,	Y =   -392.795  mm,	Z =   -246.813  mm,
	W =  90.000 deg,	P =   0.000 deg,	R =   90.000 deg
};
P[515]{
   GP1:
	UF : 0, UT : 6,		CONFIG : 'N U T, 0, 0, 0',
	X =  232.059  mm,	Y =   -391.913  mm,	Z =   -246.872  mm,
	W =  90.000 deg,	P =   0.000 deg,	R =   90.000 deg
};
P[516]{
   GP1:
	UF : 0, UT : 6,		CONFIG : 'N U T, 0, 0, 0',
	X =  234.963  mm,	Y =   -390.247  mm,	Z =   -246.744  mm,
	W =  90.000 deg,	P =   0.000 deg,	R =   90.000 deg
};
P[517]{
   GP1:
	UF : 0, UT : 6,		CONFIG : 'N U T, 0, 0, 0',
	X =  235.829  mm,	Y =   -389.736  mm,	Z =   -246.875  mm,
	W =  90.000 deg,	P =   0.000 deg,	R =   90.000 deg
};
P[518]{
   GP1:
	UF : 0, UT : 6,		CONFIG : 'N U T, 0, 0, 0',
	X =  238.638  mm,	Y =   -388.110  mm,	Z =   -246.922  mm,
	W =  90.000 deg,	P =   0.000 deg,	R =   90.000 deg
};
P[519]{
   GP1:
	UF : 0, UT : 6,		CONFIG : 'N U T, 0, 0, 0',
	X =  240.145  mm,	Y =   -387.242  mm,	Z =   -246.900  mm,
	W =  90.000 deg,	P =   0.000 deg,	R =   90.000 deg
};
P[520]{
   GP1:
	UF : 0, UT : 6,		CONFIG : 'N U T, 0, 0, 0',
	X =  241.537  mm,	Y =   -386.446  mm,	Z =   -246.810  mm,
	W =  90.000 deg,	P =   0.000 deg,	R =   90.000 deg
};
P[521]{
   GP1:
	UF : 0, UT : 6,		CONFIG : 'N U T, 0, 0, 0',
	X =  242.310  mm,	Y =   -385.991  mm,	Z =   -246.918  mm,
	W =  90.000 deg,	P =   0.000 deg,	R =   90.000 deg
};
P[522]{
   GP1:
	UF : 0, UT : 6,		CONFIG : 'N U T, 0, 0, 0',
	X =  243.125  mm,	Y =   -385.527  mm,	Z =   -246.827  mm,
	W =  90.000 deg,	P =   0.000 deg,	R =   90.000 deg
};
P[523]{
   GP1:
	UF : 0, UT : 6,		CONFIG : 'N U T, 0, 0, 0',
	X =  245.202  mm,	Y =   -384.321  mm,	Z =   -246.920  mm,
	W =  90.000 deg,	P =   0.000 deg,	R =   90.000 deg
};
P[524]{
   GP1:
	UF : 0, UT : 6,		CONFIG : 'N U T, 0, 0, 0',
	X =  248.936  mm,	Y =   -382.167  mm,	Z =   -246.892  mm,
	W =  90.000 deg,	P =   0.000 deg,	R =   90.000 deg
};
P[525]{
   GP1:
	UF : 0, UT : 6,		CONFIG : 'N U T, 0, 0, 0',
	X =  252.632  mm,	Y =   -380.029  mm,	Z =   -246.937  mm,
	W =  90.000 deg,	P =   0.000 deg,	R =   90.000 deg
};
P[526]{
   GP1:
	UF : 0, UT : 6,		CONFIG : 'N U T, 0, 0, 0',
	X =  254.141  mm,	Y =   -379.160  mm,	Z =   -246.914  mm,
	W =  90.000 deg,	P =   0.000 deg,	R =   90.000 deg
};
P[527]{
   GP1:
	UF : 0, UT : 6,		CONFIG : 'N U T, 0, 0, 0',
	X =  254.810  mm,	Y =   -378.781  mm,	Z =   -246.831  mm,
	W =  90.000 deg,	P =   0.000 deg,	R =   90.000 deg
};
P[528]{
   GP1:
	UF : 0, UT : 6,		CONFIG : 'N U T, 0, 0, 0',
	X =  255.619  mm,	Y =   -378.305  mm,	Z =   -246.943  mm,
	W =  90.000 deg,	P =   0.000 deg,	R =   90.000 deg
};
P[529]{
   GP1:
	UF : 0, UT : 6,		CONFIG : 'N U T, 0, 0, 0',
	X =  257.023  mm,	Y =   -377.498  mm,	Z =   -246.885  mm,
	W =  90.000 deg,	P =   0.000 deg,	R =   90.000 deg
};
P[530]{
   GP1:
	UF : 0, UT : 6,		CONFIG : 'N U T, 0, 0, 0',
	X =  259.978  mm,	Y =   -375.793  mm,	Z =   -246.878  mm,
	W =  90.000 deg,	P =   0.000 deg,	R =   90.000 deg
};
P[531]{
   GP1:
	UF : 0, UT : 6,		CONFIG : 'N U T, 0, 0, 0',
	X =  261.406  mm,	Y =   -374.969  mm,	Z =   -246.864  mm,
	W =  90.000 deg,	P =   0.000 deg,	R =   90.000 deg
};
P[532]{
   GP1:
	UF : 0, UT : 6,		CONFIG : 'N U T, 0, 0, 0',
	X =  262.259  mm,	Y =   -374.476  mm,	Z =   -246.874  mm,
	W =  90.000 deg,	P =   0.000 deg,	R =   90.000 deg
};
P[533]{
   GP1:
	UF : 0, UT : 6,		CONFIG : 'N U T, 0, 0, 0',
	X =  263.137  mm,	Y =   -373.971  mm,	Z =   -246.854  mm,
	W =  90.000 deg,	P =   0.000 deg,	R =   90.000 deg
};
P[534]{
   GP1:
	UF : 0, UT : 6,		CONFIG : 'N U T, 0, 0, 0',
	X =  264.442  mm,	Y =   -373.211  mm,	Z =   -246.931  mm,
	W =  90.000 deg,	P =   0.000 deg,	R =   90.000 deg
};
P[535]{
   GP1:
	UF : 0, UT : 6,		CONFIG : 'N U T, 0, 0, 0',
	X =  265.226  mm,	Y =   -372.772  mm,	Z =   -246.770  mm,
	W =  90.000 deg,	P =   0.000 deg,	R =   90.000 deg
};
P[536]{
   GP1:
	UF : 0, UT : 6,		CONFIG : 'N U T, 0, 0, 0',
	X =  266.695  mm,	Y =   -371.911  mm,	Z =   -246.923  mm,
	W =  90.000 deg,	P =   0.000 deg,	R =   90.000 deg
};
P[537]{
   GP1:
	UF : 0, UT : 6,		CONFIG : 'N U T, 0, 0, 0',
	X =  269.583  mm,	Y =   -370.139  mm,	Z =   -246.904  mm,
	W =  90.000 deg,	P =   0.000 deg,	R =   90.000 deg
};
P[538]{
   GP1:
	UF : 0, UT : 6,		CONFIG : 'N U T, 0, 0, 0',
	X =  271.378  mm,	Y =   -368.260  mm,	Z =   -246.875  mm,
	W =  90.000 deg,	P =   0.000 deg,	R =   90.000 deg
};
P[539]{
   GP1:
	UF : 0, UT : 6,		CONFIG : 'N U T, 0, 0, 0',
	X =  271.891  mm,	Y =   -367.421  mm,	Z =   -246.828  mm,
	W =  90.000 deg,	P =   0.000 deg,	R =   90.000 deg
};
P[540]{
   GP1:
	UF : 0, UT : 6,		CONFIG : 'N U T, 0, 0, 0',
	X =  272.219  mm,	Y =   -366.745  mm,	Z =   -246.768  mm,
	W =  90.000 deg,	P =   0.000 deg,	R =   90.000 deg
};
P[541]{
   GP1:
	UF : 0, UT : 6,		CONFIG : 'N U T, 0, 0, 0',
	X =  272.577  mm,	Y =   -365.700  mm,	Z =   -246.845  mm,
	W =  90.000 deg,	P =   0.000 deg,	R =   90.000 deg
};
P[542]{
   GP1:
	UF : 0, UT : 6,		CONFIG : 'N U T, 0, 0, 0',
	X =  272.877  mm,	Y =   -363.792  mm,	Z =   -246.895  mm,
	W =  90.000 deg,	P =   0.000 deg,	R =   90.000 deg
};
P[543]{
   GP1:
	UF : 0, UT : 6,		CONFIG : 'N U T, 0, 0, 0',
	X =  272.861  mm,	Y =   -362.725  mm,	Z =   -246.788  mm,
	W =  90.000 deg,	P =   0.000 deg,	R =   90.000 deg
};
P[544]{
   GP1:
	UF : 0, UT : 6,		CONFIG : 'N U T, 0, 0, 0',
	X =  272.716  mm,	Y =   -361.771  mm,	Z =   -246.913  mm,
	W =  90.000 deg,	P =   0.000 deg,	R =   90.000 deg
};
P[545]{
   GP1:
	UF : 0, UT : 6,		CONFIG : 'N U T, 0, 0, 0',
	X =  272.548  mm,	Y =   -361.057  mm,	Z =   -246.802  mm,
	W =  90.000 deg,	P =   0.000 deg,	R =   90.000 deg
};
P[546]{
   GP1:
	UF : 0, UT : 6,		CONFIG : 'N U T, 0, 0, 0',
	X =  272.465  mm,	Y =   -360.718  mm,	Z =   -246.516  mm,
	W =  90.000 deg,	P =   0.000 deg,	R =   90.000 deg
};
P[547]{
   GP1:
	UF : 0, UT : 6,		CONFIG : 'N U T, 0, 0, 0',
	X =  272.220  mm,	Y =   -360.156  mm,	Z =   -246.935  mm,
	W =  90.000 deg,	P =   0.000 deg,	R =   90.000 deg
};
P[548]{
   GP1:
	UF : 0, UT : 6,		CONFIG : 'N U T, 0, 0, 0',
	X =  271.896  mm,	Y =   -359.461  mm,	Z =   -246.843  mm,
	W =  90.000 deg,	P =   0.000 deg,	R =   90.000 deg
};
P[549]{
   GP1:
	UF : 0, UT : 6,		CONFIG : 'N U T, 0, 0, 0',
	X =  270.204  mm,	Y =   -356.498  mm,	Z =   -246.931  mm,
	W =  90.000 deg,	P =   0.000 deg,	R =   90.000 deg
};
P[550]{
   GP1:
	UF : 0, UT : 6,		CONFIG : 'N U T, 0, 0, 0',
	X =  269.796  mm,	Y =   -355.789  mm,	Z =   -246.910  mm,
	W =  90.000 deg,	P =   0.000 deg,	R =   90.000 deg
};
P[551]{
   GP1:
	UF : 0, UT : 6,		CONFIG : 'N U T, 0, 0, 0',
	X =  269.312  mm,	Y =   -354.956  mm,	Z =   -246.942  mm,
	W =  90.000 deg,	P =   0.000 deg,	R =   90.000 deg
};
P[552]{
   GP1:
	UF : 0, UT : 6,		CONFIG : 'N U T, 0, 0, 0',
	X =  268.457  mm,	Y =   -353.457  mm,	Z =   -246.828  mm,
	W =  90.000 deg,	P =   0.000 deg,	R =   90.000 deg
};
P[553]{
   GP1:
	UF : 0, UT : 6,		CONFIG : 'N U T, 0, 0, 0',
	X =  268.006  mm,	Y =   -352.680  mm,	Z =   -246.845  mm,
	W =  90.000 deg,	P =   0.000 deg,	R =   90.000 deg
};
P[554]{
   GP1:
	UF : 0, UT : 6,		CONFIG : 'N U T, 0, 0, 0',
	X =  266.774  mm,	Y =   -350.559  mm,	Z =   -246.940  mm,
	W =  90.000 deg,	P =   0.000 deg,	R =   90.000 deg
};
P[555]{
   GP1:
	UF : 0, UT : 6,		CONFIG : 'N U T, 0, 0, 0',
	X =  266.329  mm,	Y =   -349.785  mm,	Z =   -246.919  mm,
	W =  90.000 deg,	P =   0.000 deg,	R =   90.000 deg
};
P[556]{
   GP1:
	UF : 0, UT : 6,		CONFIG : 'N U T, 0, 0, 0',
	X =  265.452  mm,	Y =   -348.264  mm,	Z =   -246.908  mm,
	W =  90.000 deg,	P =   0.000 deg,	R =   90.000 deg
};
P[557]{
   GP1:
	UF : 0, UT : 6,		CONFIG : 'N U T, 0, 0, 0',
	X =  265.062  mm,	Y =   -347.594  mm,	Z =   -246.943  mm,
	W =  90.000 deg,	P =   0.000 deg,	R =   90.000 deg
};
P[558]{
   GP1:
	UF : 0, UT : 6,		CONFIG : 'N U T, 0, 0, 0',
	X =  264.604  mm,	Y =   -346.796  mm,	Z =   -246.915  mm,
	W =  90.000 deg,	P =   0.000 deg,	R =   90.000 deg
};
P[559]{
   GP1:
	UF : 0, UT : 6,		CONFIG : 'N U T, 0, 0, 0',
	X =  264.199  mm,	Y =   -346.093  mm,	Z =   -246.903  mm,
	W =  90.000 deg,	P =   0.000 deg,	R =   90.000 deg
};
P[560]{
   GP1:
	UF : 0, UT : 6,		CONFIG : 'N U T, 0, 0, 0',
	X =  261.658  mm,	Y =   -341.694  mm,	Z =   -246.909  mm,
	W =  90.000 deg,	P =   0.000 deg,	R =   90.000 deg
};
P[561]{
   GP1:
	UF : 0, UT : 6,		CONFIG : 'N U T, 0, 0, 0',
	X =  261.275  mm,	Y =   -341.009  mm,	Z =   -246.762  mm,
	W =  90.000 deg,	P =   0.000 deg,	R =   90.000 deg
};
P[562]{
   GP1:
	UF : 0, UT : 6,		CONFIG : 'N U T, 0, 0, 0',
	X =  260.384  mm,	Y =   -339.475  mm,	Z =   -246.813  mm,
	W =  90.000 deg,	P =   0.000 deg,	R =   90.000 deg
};
P[563]{
   GP1:
	UF : 0, UT : 6,		CONFIG : 'N U T, 0, 0, 0',
	X =  259.930  mm,	Y =   -338.701  mm,	Z =   -246.911  mm,
	W =  90.000 deg,	P =   0.000 deg,	R =   90.000 deg
};
P[564]{
   GP1:
	UF : 0, UT : 6,		CONFIG : 'N U T, 0, 0, 0',
	X =  259.531  mm,	Y =   -338.007  mm,	Z =   -246.884  mm,
	W =  90.000 deg,	P =   0.000 deg,	R =   90.000 deg
};
P[565]{
   GP1:
	UF : 0, UT : 6,		CONFIG : 'N U T, 0, 0, 0',
	X =  257.834  mm,	Y =   -335.060  mm,	Z =   -246.831  mm,
	W =  90.000 deg,	P =   0.000 deg,	R =   90.000 deg
};
P[566]{
   GP1:
	UF : 0, UT : 6,		CONFIG : 'N U T, 0, 0, 0',
	X =  257.389  mm,	Y =   -334.303  mm,	Z =   -246.924  mm,
	W =  90.000 deg,	P =   0.000 deg,	R =   90.000 deg
};
P[567]{
   GP1:
	UF : 0, UT : 6,		CONFIG : 'N U T, 0, 0, 0',
	X =  256.103  mm,	Y =   -332.071  mm,	Z =   -246.894  mm,
	W =  90.000 deg,	P =   0.000 deg,	R =   90.000 deg
};
P[568]{
   GP1:
	UF : 0, UT : 6,		CONFIG : 'N U T, 0, 0, 0',
	X =  255.217  mm,	Y =   -330.533  mm,	Z =   -246.868  mm,
	W =  90.000 deg,	P =   0.000 deg,	R =   90.000 deg
};
P[569]{
   GP1:
	UF : 0, UT : 6,		CONFIG : 'N U T, 0, 0, 0',
	X =  254.844  mm,	Y =   -329.885  mm,	Z =   -246.855  mm,
	W =  90.000 deg,	P =   0.000 deg,	R =   90.000 deg
};
P[570]{
   GP1:
	UF : 0, UT : 6,		CONFIG : 'N U T, 0, 0, 0',
	X =  254.459  mm,	Y =   -329.250  mm,	Z =   -246.891  mm,
	W =  90.000 deg,	P =   0.000 deg,	R =   90.000 deg
};
P[571]{
   GP1:
	UF : 0, UT : 6,		CONFIG : 'N U T, 0, 0, 0',
	X =  254.017  mm,	Y =   -328.595  mm,	Z =   -246.865  mm,
	W =  90.000 deg,	P =   0.000 deg,	R =   90.000 deg
};
P[572]{
   GP1:
	UF : 0, UT : 6,		CONFIG : 'N U T, 0, 0, 0',
	X =  253.659  mm,	Y =   -328.139  mm,	Z =   -246.750  mm,
	W =  90.000 deg,	P =   0.000 deg,	R =   90.000 deg
};
P[573]{
   GP1:
	UF : 0, UT : 6,		CONFIG : 'N U T, 0, 0, 0',
	X =  253.332  mm,	Y =   -327.789  mm,	Z =   -246.838  mm,
	W =  90.000 deg,	P =   0.000 deg,	R =   90.000 deg
};
P[574]{
   GP1:
	UF : 0, UT : 6,		CONFIG : 'N U T, 0, 0, 0',
	X =  252.893  mm,	Y =   -327.355  mm,	Z =   -246.826  mm,
	W =  90.000 deg,	P =   0.000 deg,	R =   90.000 deg
};
P[575]{
   GP1:
	UF : 0, UT : 6,		CONFIG : 'N U T, 0, 0, 0',
	X =  251.172  mm,	Y =   -326.156  mm,	Z =   -246.831  mm,
	W =  90.000 deg,	P =   0.000 deg,	R =   90.000 deg
};
P[576]{
   GP1:
	UF : 0, UT : 6,		CONFIG : 'N U T, 0, 0, 0',
	X =  248.832  mm,	Y =   -325.323  mm,	Z =   -246.778  mm,
	W =  90.000 deg,	P =   0.000 deg,	R =   90.000 deg
};
P[577]{
   GP1:
	UF : 0, UT : 6,		CONFIG : 'N U T, 0, 0, 0',
	X =  244.810  mm,	Y =   -325.540  mm,	Z =   -246.864  mm,
	W =  90.000 deg,	P =   0.000 deg,	R =   90.000 deg
};
P[578]{
   GP1:
	UF : 0, UT : 6,		CONFIG : 'N U T, 0, 0, 0',
	X =  244.473  mm,	Y =   -325.624  mm,	Z =   -246.590  mm,
	W =  90.000 deg,	P =   0.000 deg,	R =   90.000 deg
};
P[579]{
   GP1:
	UF : 0, UT : 6,		CONFIG : 'N U T, 0, 0, 0',
	X =  243.237  mm,	Y =   -326.183  mm,	Z =   -246.868  mm,
	W =  90.000 deg,	P =   0.000 deg,	R =   90.000 deg
};
P[580]{
   GP1:
	UF : 0, UT : 6,		CONFIG : 'N U T, 0, 0, 0',
	X =  240.384  mm,	Y =   -327.804  mm,	Z =   -246.837  mm,
	W =  90.000 deg,	P =   0.000 deg,	R =   90.000 deg
};
P[581]{
   GP1:
	UF : 0, UT : 6,		CONFIG : 'N U T, 0, 0, 0',
	X =  239.545  mm,	Y =   -328.287  mm,	Z =   -246.828  mm,
	W =  90.000 deg,	P =   0.000 deg,	R =   90.000 deg
};
P[582]{
   GP1:
	UF : 0, UT : 6,		CONFIG : 'N U T, 0, 0, 0',
	X =  237.324  mm,	Y =   -329.574  mm,	Z =   -246.875  mm,
	W =  90.000 deg,	P =   0.000 deg,	R =   90.000 deg
};
P[583]{
   GP1:
	UF : 0, UT : 6,		CONFIG : 'N U T, 0, 0, 0',
	X =  235.113  mm,	Y =   -330.855  mm,	Z =   -246.935  mm,
	W =  90.000 deg,	P =   0.000 deg,	R =   90.000 deg
};
P[584]{
   GP1:
	UF : 0, UT : 6,		CONFIG : 'N U T, 0, 0, 0',
	X =  234.371  mm,	Y =   -331.275  mm,	Z =   -246.838  mm,
	W =  90.000 deg,	P =   0.000 deg,	R =   90.000 deg
};
P[585]{
   GP1:
	UF : 0, UT : 6,		CONFIG : 'N U T, 0, 0, 0',
	X =  233.586  mm,	Y =   -331.729  mm,	Z =   -246.847  mm,
	W =  90.000 deg,	P =   0.000 deg,	R =   90.000 deg
};
P[586]{
   GP1:
	UF : 0, UT : 6,		CONFIG : 'N U T, 0, 0, 0',
	X =  232.764  mm,	Y =   -332.210  mm,	Z =   -246.922  mm,
	W =  90.000 deg,	P =   0.000 deg,	R =   90.000 deg
};
P[587]{
   GP1:
	UF : 0, UT : 6,		CONFIG : 'N U T, 0, 0, 0',
	X =  226.921  mm,	Y =   -335.581  mm,	Z =   -246.893  mm,
	W =  90.000 deg,	P =   0.000 deg,	R =   90.000 deg
};
P[588]{
   GP1:
	UF : 0, UT : 6,		CONFIG : 'N U T, 0, 0, 0',
	X =  224.739  mm,	Y =   -336.844  mm,	Z =   -246.931  mm,
	W =  90.000 deg,	P =   0.000 deg,	R =   90.000 deg
};
P[589]{
   GP1:
	UF : 0, UT : 6,		CONFIG : 'N U T, 0, 0, 0',
	X =  221.162  mm,	Y =   -338.911  mm,	Z =   -246.941  mm,
	W =  90.000 deg,	P =   0.000 deg,	R =   90.000 deg
};
P[590]{
   GP1:
	UF : 0, UT : 6,		CONFIG : 'N U T, 0, 0, 0',
	X =  219.593  mm,	Y =   -339.816  mm,	Z =   -246.930  mm,
	W =  90.000 deg,	P =   0.000 deg,	R =   90.000 deg
};
P[591]{
   GP1:
	UF : 0, UT : 6,		CONFIG : 'N U T, 0, 0, 0',
	X =  218.974  mm,	Y =   -340.173  mm,	Z =   -246.934  mm,
	W =  90.000 deg,	P =   0.000 deg,	R =   90.000 deg
};
P[592]{
   GP1:
	UF : 0, UT : 6,		CONFIG : 'N U T, 0, 0, 0',
	X =  218.235  mm,	Y =   -340.588  mm,	Z =   -246.783  mm,
	W =  90.000 deg,	P =   0.000 deg,	R =   90.000 deg
};
P[593]{
   GP1:
	UF : 0, UT : 6,		CONFIG : 'N U T, 0, 0, 0',
	X =  216.662  mm,	Y =   -341.507  mm,	Z =   -246.919  mm,
	W =  90.000 deg,	P =   0.000 deg,	R =   90.000 deg
};
P[594]{
   GP1:
	UF : 0, UT : 6,		CONFIG : 'N U T, 0, 0, 0',
	X =  215.924  mm,	Y =   -341.926  mm,	Z =   -246.830  mm,
	W =  90.000 deg,	P =   0.000 deg,	R =   90.000 deg
};
P[595]{
   GP1:
	UF : 0, UT : 6,		CONFIG : 'N U T, 0, 0, 0',
	X =  213.876  mm,	Y =   -343.114  mm,	Z =   -246.902  mm,
	W =  90.000 deg,	P =   0.000 deg,	R =   90.000 deg
};
P[596]{
   GP1:
	UF : 0, UT : 6,		CONFIG : 'N U T, 0, 0, 0',
	X =  212.197  mm,	Y =   -344.080  mm,	Z =   -246.854  mm,
	W =  90.000 deg,	P =   0.000 deg,	R =   90.000 deg
};
P[597]{
   GP1:
	UF : 0, UT : 6,		CONFIG : 'N U T, 0, 0, 0',
	X =  211.506  mm,	Y =   -344.476  mm,	Z =   -246.821  mm,
	W =  90.000 deg,	P =   0.000 deg,	R =   90.000 deg
};
P[598]{
   GP1:
	UF : 0, UT : 6,		CONFIG : 'N U T, 0, 0, 0',
	X =  210.054  mm,	Y =   -345.321  mm,	Z =   -246.902  mm,
	W =  90.000 deg,	P =   0.000 deg,	R =   90.000 deg
};
P[599]{
   GP1:
	UF : 0, UT : 6,		CONFIG : 'N U T, 0, 0, 0',
	X =  205.705  mm,	Y =   -347.832  mm,	Z =   -246.899  mm,
	W =  90.000 deg,	P =   0.000 deg,	R =   90.000 deg
};
P[600]{
   GP1:
	UF : 0, UT : 6,		CONFIG : 'N U T, 0, 0, 0',
	X =  204.132  mm,	Y =   -348.737  mm,	Z =   -246.857  mm,
	W =  90.000 deg,	P =   0.000 deg,	R =   90.000 deg
};
P[601]{
   GP1:
	UF : 0, UT : 6,		CONFIG : 'N U T, 0, 0, 0',
	X =  203.491  mm,	Y =   -349.105  mm,	Z =   -246.837  mm,
	W =  90.000 deg,	P =   0.000 deg,	R =   90.000 deg
};
P[602]{
   GP1:
	UF : 0, UT : 6,		CONFIG : 'N U T, 0, 0, 0',
	X =  202.758  mm,	Y =   -349.535  mm,	Z =   -246.914  mm,
	W =  90.000 deg,	P =   0.000 deg,	R =   90.000 deg
};
P[603]{
   GP1:
	UF : 0, UT : 6,		CONFIG : 'N U T, 0, 0, 0',
	X =  199.775  mm,	Y =   -351.249  mm,	Z =   -246.813  mm,
	W =  90.000 deg,	P =   0.000 deg,	R =   90.000 deg
};
P[604]{
   GP1:
	UF : 0, UT : 6,		CONFIG : 'N U T, 0, 0, 0',
	X =  198.231  mm,	Y =   -352.144  mm,	Z =   -246.859  mm,
	W =  90.000 deg,	P =   0.000 deg,	R =   90.000 deg
};
P[605]{
   GP1:
	UF : 0, UT : 6,		CONFIG : 'N U T, 0, 0, 0',
	X =  197.528  mm,	Y =   -352.555  mm,	Z =   -246.923  mm,
	W =  90.000 deg,	P =   0.000 deg,	R =   90.000 deg
};
P[606]{
   GP1:
	UF : 0, UT : 6,		CONFIG : 'N U T, 0, 0, 0',
	X =  196.452  mm,	Y =   -352.414  mm,	Z =   -237.472  mm,
	W =  90.000 deg,	P =   0.000 deg,	R =   90.000 deg
};
P[607]{
   GP1:
	UF : 0, UT : 6,		CONFIG : 'N U T, 0, 0, 0',
	X =  195.593  mm,	Y =   -352.912  mm,	Z =   -237.503  mm,
	W =  90.000 deg,	P =   0.000 deg,	R =   90.000 deg
};
P[608]{
   GP1:
	UF : 0, UT : 6,		CONFIG : 'N U T, 0, 0, 0',
	X =  194.880  mm,	Y =   -353.320  mm,	Z =   -237.459  mm,
	W =  90.000 deg,	P =   0.000 deg,	R =   90.000 deg
};
P[609]{
   GP1:
	UF : 0, UT : 6,		CONFIG : 'N U T, 0, 0, 0',
	X =  194.361  mm,	Y =   -353.624  mm,	Z =   -237.503  mm,
	W =  90.000 deg,	P =   0.000 deg,	R =   90.000 deg
};
P[610]{
   GP1:
	UF : 0, UT : 6,		CONFIG : 'N U T, 0, 0, 0',
	X =  192.742  mm,	Y =   -354.554  mm,	Z =   -237.452  mm,
	W =  90.000 deg,	P =   0.000 deg,	R =   90.000 deg
};
P[611]{
   GP1:
	UF : 0, UT : 6,		CONFIG : 'N U T, 0, 0, 0',
	X =  192.213  mm,	Y =   -354.834  mm,	Z =   -237.137  mm,
	W =  90.000 deg,	P =   0.000 deg,	R =   90.000 deg
};
P[612]{
   GP1:
	UF : 0, UT : 6,		CONFIG : 'N U T, 0, 0, 0',
	X =  192.054  mm,	Y =   -354.961  mm,	Z =   -237.577  mm,
	W =  90.000 deg,	P =   0.000 deg,	R =   90.000 deg
};
P[613]{
   GP1:
	UF : 0, UT : 6,		CONFIG : 'N U T, 0, 0, 0',
	X =  191.526  mm,	Y =   -355.232  mm,	Z =   -237.155  mm,
	W =  90.000 deg,	P =   0.000 deg,	R =   90.000 deg
};
P[614]{
   GP1:
	UF : 0, UT : 6,		CONFIG : 'N U T, 0, 0, 0',
	X =  191.288  mm,	Y =   -355.402  mm,	Z =   -237.566  mm,
	W =  90.000 deg,	P =   0.000 deg,	R =   90.000 deg
};
P[615]{
   GP1:
	UF : 0, UT : 6,		CONFIG : 'N U T, 0, 0, 0',
	X =  189.876  mm,	Y =   -356.219  mm,	Z =   -237.579  mm,
	W =  90.000 deg,	P =   0.000 deg,	R =   90.000 deg
};
P[616]{
   GP1:
	UF : 0, UT : 6,		CONFIG : 'N U T, 0, 0, 0',
	X =  189.605  mm,	Y =   -356.340  mm,	Z =   -237.141  mm,
	W =  90.000 deg,	P =   0.000 deg,	R =   90.000 deg
};
P[617]{
   GP1:
	UF : 0, UT : 6,		CONFIG : 'N U T, 0, 0, 0',
	X =  189.093  mm,	Y =   -356.670  mm,	Z =   -237.570  mm,
	W =  90.000 deg,	P =   0.000 deg,	R =   90.000 deg
};
P[618]{
   GP1:
	UF : 0, UT : 6,		CONFIG : 'N U T, 0, 0, 0',
	X =  188.357  mm,	Y =   -357.097  mm,	Z =   -237.589  mm,
	W =  90.000 deg,	P =   0.000 deg,	R =   90.000 deg
};
P[619]{
   GP1:
	UF : 0, UT : 6,		CONFIG : 'N U T, 0, 0, 0',
	X =  186.886  mm,	Y =   -357.936  mm,	Z =   -237.464  mm,
	W =  90.000 deg,	P =   0.000 deg,	R =   90.000 deg
};
P[620]{
   GP1:
	UF : 0, UT : 6,		CONFIG : 'N U T, 0, 0, 0',
	X =  185.815  mm,	Y =   -358.527  mm,	Z =   -237.125  mm,
	W =  90.000 deg,	P =   0.000 deg,	R =   90.000 deg
};
P[621]{
   GP1:
	UF : 0, UT : 6,		CONFIG : 'N U T, 0, 0, 0',
	X =  183.926  mm,	Y =   -359.647  mm,	Z =   -237.479  mm,
	W =  90.000 deg,	P =   0.000 deg,	R =   90.000 deg
};
P[622]{
   GP1:
	UF : 0, UT : 6,		CONFIG : 'N U T, 0, 0, 0',
	X =  183.331  mm,	Y =   -359.961  mm,	Z =   -237.119  mm,
	W =  90.000 deg,	P =   0.000 deg,	R =   90.000 deg
};
P[623]{
   GP1:
	UF : 0, UT : 6,		CONFIG : 'N U T, 0, 0, 0',
	X =  183.210  mm,	Y =   -360.063  mm,	Z =   -237.525  mm,
	W =  90.000 deg,	P =   0.000 deg,	R =   90.000 deg
};
P[624]{
   GP1:
	UF : 0, UT : 6,		CONFIG : 'N U T, 0, 0, 0',
	X =  180.716  mm,	Y =   -361.473  mm,	Z =   -237.142  mm,
	W =  90.000 deg,	P =   0.000 deg,	R =   90.000 deg
};
P[625]{
   GP1:
	UF : 0, UT : 6,		CONFIG : 'N U T, 0, 0, 0',
	X =  179.430  mm,	Y =   -362.216  mm,	Z =   -237.155  mm,
	W =  90.000 deg,	P =   0.000 deg,	R =   90.000 deg
};
P[626]{
   GP1:
	UF : 0, UT : 6,		CONFIG : 'N U T, 0, 0, 0',
	X =  178.677  mm,	Y =   -362.681  mm,	Z =   -237.526  mm,
	W =  90.000 deg,	P =   0.000 deg,	R =   90.000 deg
};
P[627]{
   GP1:
	UF : 0, UT : 6,		CONFIG : 'N U T, 0, 0, 0',
	X =  176.684  mm,	Y =   -363.827  mm,	Z =   -237.472  mm,
	W =  90.000 deg,	P =   0.000 deg,	R =   90.000 deg
};
P[628]{
   GP1:
	UF : 0, UT : 6,		CONFIG : 'N U T, 0, 0, 0',
	X =  175.124  mm,	Y =   -364.735  mm,	Z =   -237.561  mm,
	W =  90.000 deg,	P =   0.000 deg,	R =   90.000 deg
};
P[629]{
   GP1:
	UF : 0, UT : 6,		CONFIG : 'N U T, 0, 0, 0',
	X =  174.385  mm,	Y =   -365.161  mm,	Z =   -237.543  mm,
	W =  90.000 deg,	P =   0.000 deg,	R =   90.000 deg
};
P[630]{
   GP1:
	UF : 0, UT : 6,		CONFIG : 'N U T, 0, 0, 0',
	X =  173.689  mm,	Y =   -365.562  mm,	Z =   -237.543  mm,
	W =  90.000 deg,	P =   0.000 deg,	R =   90.000 deg
};
P[631]{
   GP1:
	UF : 0, UT : 6,		CONFIG : 'N U T, 0, 0, 0',
	X =  171.462  mm,	Y =   -366.852  mm,	Z =   -237.587  mm,
	W =  90.000 deg,	P =   0.000 deg,	R =   90.000 deg
};
P[632]{
   GP1:
	UF : 0, UT : 6,		CONFIG : 'N U T, 0, 0, 0',
	X =  170.757  mm,	Y =   -367.254  mm,	Z =   -237.523  mm,
	W =  90.000 deg,	P =   0.000 deg,	R =   90.000 deg
};
P[633]{
   GP1:
	UF : 0, UT : 6,		CONFIG : 'N U T, 0, 0, 0',
	X =  168.797  mm,	Y =   -368.355  mm,	Z =   -237.147  mm,
	W =  90.000 deg,	P =   0.000 deg,	R =   90.000 deg
};
P[634]{
   GP1:
	UF : 0, UT : 6,		CONFIG : 'N U T, 0, 0, 0',
	X =  167.771  mm,	Y =   -368.983  mm,	Z =   -237.590  mm,
	W =  90.000 deg,	P =   0.000 deg,	R =   90.000 deg
};
P[635]{
   GP1:
	UF : 0, UT : 6,		CONFIG : 'N U T, 0, 0, 0',
	X =  167.226  mm,	Y =   -369.262  mm,	Z =   -237.146  mm,
	W =  90.000 deg,	P =   0.000 deg,	R =   90.000 deg
};
P[636]{
   GP1:
	UF : 0, UT : 6,		CONFIG : 'N U T, 0, 0, 0',
	X =  167.006  mm,	Y =   -369.423  mm,	Z =   -237.569  mm,
	W =  90.000 deg,	P =   0.000 deg,	R =   90.000 deg
};
P[637]{
   GP1:
	UF : 0, UT : 6,		CONFIG : 'N U T, 0, 0, 0',
	X =  166.316  mm,	Y =   -369.815  mm,	Z =   -237.492  mm,
	W =  90.000 deg,	P =   0.000 deg,	R =   90.000 deg
};
P[638]{
   GP1:
	UF : 0, UT : 6,		CONFIG : 'N U T, 0, 0, 0',
	X =  165.597  mm,	Y =   -370.229  mm,	Z =   -237.469  mm,
	W =  90.000 deg,	P =   0.000 deg,	R =   90.000 deg
};
P[639]{
   GP1:
	UF : 0, UT : 6,		CONFIG : 'N U T, 0, 0, 0',
	X =  163.993  mm,	Y =   -371.160  mm,	Z =   -237.536  mm,
	W =  90.000 deg,	P =   0.000 deg,	R =   90.000 deg
};
P[640]{
   GP1:
	UF : 0, UT : 6,		CONFIG : 'N U T, 0, 0, 0',
	X =  162.510  mm,	Y =   -372.014  mm,	Z =   -237.501  mm,
	W =  90.000 deg,	P =   0.000 deg,	R =   90.000 deg
};
P[641]{
   GP1:
	UF : 0, UT : 6,		CONFIG : 'N U T, 0, 0, 0',
	X =  161.068  mm,	Y =   -372.816  mm,	Z =   -237.118  mm,
	W =  90.000 deg,	P =   0.000 deg,	R =   90.000 deg
};
P[642]{
   GP1:
	UF : 0, UT : 6,		CONFIG : 'N U T, 0, 0, 0',
	X =  161.103  mm,	Y =   -372.832  mm,	Z =   -237.573  mm,
	W =  90.000 deg,	P =   0.000 deg,	R =   90.000 deg
};
P[643]{
   GP1:
	UF : 0, UT : 6,		CONFIG : 'N U T, 0, 0, 0',
	X =  160.340  mm,	Y =   -373.267  mm,	Z =   -237.510  mm,
	W =  90.000 deg,	P =   0.000 deg,	R =   90.000 deg
};
P[644]{
   GP1:
	UF : 0, UT : 6,		CONFIG : 'N U T, 0, 0, 0',
	X =  158.226  mm,	Y =   -374.490  mm,	Z =   -237.532  mm,
	W =  90.000 deg,	P =   0.000 deg,	R =   90.000 deg
};
P[645]{
   GP1:
	UF : 0, UT : 6,		CONFIG : 'N U T, 0, 0, 0',
	X =  157.154  mm,	Y =   -375.077  mm,	Z =   -237.142  mm,
	W =  90.000 deg,	P =   0.000 deg,	R =   90.000 deg
};
P[646]{
   GP1:
	UF : 0, UT : 6,		CONFIG : 'N U T, 0, 0, 0',
	X =  156.872  mm,	Y =   -375.241  mm,	Z =   -237.144  mm,
	W =  90.000 deg,	P =   0.000 deg,	R =   90.000 deg
};
P[647]{
   GP1:
	UF : 0, UT : 6,		CONFIG : 'N U T, 0, 0, 0',
	X =  156.671  mm,	Y =   -375.387  mm,	Z =   -237.522  mm,
	W =  90.000 deg,	P =   0.000 deg,	R =   90.000 deg
};
P[648]{
   GP1:
	UF : 0, UT : 6,		CONFIG : 'N U T, 0, 0, 0',
	X =  156.096  mm,	Y =   -375.686  mm,	Z =   -237.118  mm,
	W =  90.000 deg,	P =   0.000 deg,	R =   90.000 deg
};
P[649]{
   GP1:
	UF : 0, UT : 6,		CONFIG : 'N U T, 0, 0, 0',
	X =  155.935  mm,	Y =   -375.811  mm,	Z =   -237.518  mm,
	W =  90.000 deg,	P =   0.000 deg,	R =   90.000 deg
};
P[650]{
   GP1:
	UF : 0, UT : 6,		CONFIG : 'N U T, 0, 0, 0',
	X =  155.262  mm,	Y =   -376.202  mm,	Z =   -237.551  mm,
	W =  90.000 deg,	P =   0.000 deg,	R =   90.000 deg
};
P[651]{
   GP1:
	UF : 0, UT : 6,		CONFIG : 'N U T, 0, 0, 0',
	X =  154.483  mm,	Y =   -376.648  mm,	Z =   -237.498  mm,
	W =  90.000 deg,	P =   0.000 deg,	R =   90.000 deg
};
P[652]{
   GP1:
	UF : 0, UT : 6,		CONFIG : 'N U T, 0, 0, 0',
	X =  152.841  mm,	Y =   -377.567  mm,	Z =   -237.130  mm,
	W =  90.000 deg,	P =   0.000 deg,	R =   90.000 deg
};
P[653]{
   GP1:
	UF : 0, UT : 6,		CONFIG : 'N U T, 0, 0, 0',
	X =  152.244  mm,	Y =   -377.911  mm,	Z =   -237.120  mm,
	W =  90.000 deg,	P =   0.000 deg,	R =   90.000 deg
};
P[654]{
   GP1:
	UF : 0, UT : 6,		CONFIG : 'N U T, 0, 0, 0',
	X =  152.246  mm,	Y =   -377.947  mm,	Z =   -237.585  mm,
	W =  90.000 deg,	P =   0.000 deg,	R =   90.000 deg
};
P[655]{
   GP1:
	UF : 0, UT : 6,		CONFIG : 'N U T, 0, 0, 0',
	X =  151.569  mm,	Y =   -378.330  mm,	Z =   -237.488  mm,
	W =  90.000 deg,	P =   0.000 deg,	R =   90.000 deg
};
P[656]{
   GP1:
	UF : 0, UT : 6,		CONFIG : 'N U T, 0, 0, 0',
	X =  150.747  mm,	Y =   -378.810  mm,	Z =   -237.557  mm,
	W =  90.000 deg,	P =   0.000 deg,	R =   90.000 deg
};
P[657]{
   GP1:
	UF : 0, UT : 6,		CONFIG : 'N U T, 0, 0, 0',
	X =  150.027  mm,	Y =   -379.269  mm,	Z =   -237.568  mm,
	W =  90.000 deg,	P =   0.000 deg,	R =   90.000 deg
};
P[658]{
   GP1:
	UF : 0, UT : 6,		CONFIG : 'N U T, 0, 0, 0',
	X =  148.119  mm,	Y =   -380.998  mm,	Z =   -237.571  mm,
	W =  90.000 deg,	P =   0.000 deg,	R =   90.000 deg
};
P[659]{
   GP1:
	UF : 0, UT : 6,		CONFIG : 'N U T, 0, 0, 0',
	X =  147.751  mm,	Y =   -381.442  mm,	Z =   -237.489  mm,
	W =  90.000 deg,	P =   0.000 deg,	R =   90.000 deg
};
P[660]{
   GP1:
	UF : 0, UT : 6,		CONFIG : 'N U T, 0, 0, 0',
	X =  147.446  mm,	Y =   -381.937  mm,	Z =   -237.469  mm,
	W =  90.000 deg,	P =   0.000 deg,	R =   90.000 deg
};
P[661]{
   GP1:
	UF : 0, UT : 6,		CONFIG : 'N U T, 0, 0, 0',
	X =  147.108  mm,	Y =   -382.565  mm,	Z =   -237.573  mm,
	W =  90.000 deg,	P =   0.000 deg,	R =   90.000 deg
};
P[662]{
   GP1:
	UF : 0, UT : 6,		CONFIG : 'N U T, 0, 0, 0',
	X =  146.239  mm,	Y =   -385.821  mm,	Z =   -237.535  mm,
	W =  90.000 deg,	P =   0.000 deg,	R =   90.000 deg
};
P[663]{
   GP1:
	UF : 0, UT : 6,		CONFIG : 'N U T, 0, 0, 0',
	X =  146.194  mm,	Y =   -386.696  mm,	Z =   -237.129  mm,
	W =  90.000 deg,	P =   0.000 deg,	R =   90.000 deg
};
P[664]{
   GP1:
	UF : 0, UT : 6,		CONFIG : 'N U T, 0, 0, 0',
	X =  146.212  mm,	Y =   -387.116  mm,	Z =   -237.215  mm,
	W =  90.000 deg,	P =   0.000 deg,	R =   90.000 deg
};
P[665]{
   GP1:
	UF : 0, UT : 6,		CONFIG : 'N U T, 0, 0, 0',
	X =  146.339  mm,	Y =   -387.692  mm,	Z =   -237.546  mm,
	W =  90.000 deg,	P =   0.000 deg,	R =   90.000 deg
};
P[666]{
   GP1:
	UF : 0, UT : 6,		CONFIG : 'N U T, 0, 0, 0',
	X =  146.498  mm,	Y =   -388.487  mm,	Z =   -237.551  mm,
	W =  90.000 deg,	P =   0.000 deg,	R =   90.000 deg
};
P[667]{
   GP1:
	UF : 0, UT : 6,		CONFIG : 'N U T, 0, 0, 0',
	X =  147.563  mm,	Y =   -390.944  mm,	Z =   -237.568  mm,
	W =  90.000 deg,	P =   0.000 deg,	R =   90.000 deg
};
P[668]{
   GP1:
	UF : 0, UT : 6,		CONFIG : 'N U T, 0, 0, 0',
	X =  148.352  mm,	Y =   -392.317  mm,	Z =   -237.517  mm,
	W =  90.000 deg,	P =   0.000 deg,	R =   90.000 deg
};
P[669]{
   GP1:
	UF : 0, UT : 6,		CONFIG : 'N U T, 0, 0, 0',
	X =  148.674  mm,	Y =   -392.930  mm,	Z =   -237.122  mm,
	W =  90.000 deg,	P =   0.000 deg,	R =   90.000 deg
};
P[670]{
   GP1:
	UF : 0, UT : 6,		CONFIG : 'N U T, 0, 0, 0',
	X =  149.676  mm,	Y =   -394.660  mm,	Z =   -237.155  mm,
	W =  90.000 deg,	P =   0.000 deg,	R =   90.000 deg
};
P[671]{
   GP1:
	UF : 0, UT : 6,		CONFIG : 'N U T, 0, 0, 0',
	X =  150.112  mm,	Y =   -395.373  mm,	Z =   -237.467  mm,
	W =  90.000 deg,	P =   0.000 deg,	R =   90.000 deg
};
P[672]{
   GP1:
	UF : 0, UT : 6,		CONFIG : 'N U T, 0, 0, 0',
	X =  150.987  mm,	Y =   -396.878  mm,	Z =   -237.541  mm,
	W =  90.000 deg,	P =   0.000 deg,	R =   90.000 deg
};
P[673]{
   GP1:
	UF : 0, UT : 6,		CONFIG : 'N U T, 0, 0, 0',
	X =  151.474  mm,	Y =   -397.779  mm,	Z =   -237.124  mm,
	W =  90.000 deg,	P =   0.000 deg,	R =   90.000 deg
};
P[674]{
   GP1:
	UF : 0, UT : 6,		CONFIG : 'N U T, 0, 0, 0',
	X =  151.786  mm,	Y =   -398.276  mm,	Z =   -237.447  mm,
	W =  90.000 deg,	P =   0.000 deg,	R =   90.000 deg
};
P[675]{
   GP1:
	UF : 0, UT : 6,		CONFIG : 'N U T, 0, 0, 0',
	X =  152.680  mm,	Y =   -399.868  mm,	Z =   -237.124  mm,
	W =  90.000 deg,	P =   0.000 deg,	R =   90.000 deg
};
P[676]{
   GP1:
	UF : 0, UT : 6,		CONFIG : 'N U T, 0, 0, 0',
	X =  153.500  mm,	Y =   -401.225  mm,	Z =   -237.580  mm,
	W =  90.000 deg,	P =   0.000 deg,	R =   90.000 deg
};
P[677]{
   GP1:
	UF : 0, UT : 6,		CONFIG : 'N U T, 0, 0, 0',
	X =  153.925  mm,	Y =   -402.023  mm,	Z =   -237.130  mm,
	W =  90.000 deg,	P =   0.000 deg,	R =   90.000 deg
};
P[678]{
   GP1:
	UF : 0, UT : 6,		CONFIG : 'N U T, 0, 0, 0',
	X =  154.294  mm,	Y =   -402.602  mm,	Z =   -237.561  mm,
	W =  90.000 deg,	P =   0.000 deg,	R =   90.000 deg
};
P[679]{
   GP1:
	UF : 0, UT : 6,		CONFIG : 'N U T, 0, 0, 0',
	X =  155.189  mm,	Y =   -404.156  mm,	Z =   -237.537  mm,
	W =  90.000 deg,	P =   0.000 deg,	R =   90.000 deg
};
P[680]{
   GP1:
	UF : 0, UT : 6,		CONFIG : 'N U T, 0, 0, 0',
	X =  156.469  mm,	Y =   -406.369  mm,	Z =   -237.562  mm,
	W =  90.000 deg,	P =   0.000 deg,	R =   90.000 deg
};
P[681]{
   GP1:
	UF : 0, UT : 6,		CONFIG : 'N U T, 0, 0, 0',
	X =  156.618  mm,	Y =   -406.686  mm,	Z =   -237.148  mm,
	W =  90.000 deg,	P =   0.000 deg,	R =   90.000 deg
};
P[682]{
   GP1:
	UF : 0, UT : 6,		CONFIG : 'N U T, 0, 0, 0',
	X =  156.925  mm,	Y =   -407.160  mm,	Z =   -237.556  mm,
	W =  90.000 deg,	P =   0.000 deg,	R =   90.000 deg
};
P[683]{
   GP1:
	UF : 0, UT : 6,		CONFIG : 'N U T, 0, 0, 0',
	X =  157.572  mm,	Y =   -408.339  mm,	Z =   -237.140  mm,
	W =  90.000 deg,	P =   0.000 deg,	R =   90.000 deg
};
P[684]{
   GP1:
	UF : 0, UT : 6,		CONFIG : 'N U T, 0, 0, 0',
	X =  158.263  mm,	Y =   -409.480  mm,	Z =   -237.535  mm,
	W =  90.000 deg,	P =   0.000 deg,	R =   90.000 deg
};
P[685]{
   GP1:
	UF : 0, UT : 6,		CONFIG : 'N U T, 0, 0, 0',
	X =  158.439  mm,	Y =   -409.844  mm,	Z =   -237.113  mm,
	W =  90.000 deg,	P =   0.000 deg,	R =   90.000 deg
};
P[686]{
   GP1:
	UF : 0, UT : 6,		CONFIG : 'N U T, 0, 0, 0',
	X =  158.665  mm,	Y =   -410.191  mm,	Z =   -237.433  mm,
	W =  90.000 deg,	P =   0.000 deg,	R =   90.000 deg
};
P[687]{
   GP1:
	UF : 0, UT : 6,		CONFIG : 'N U T, 0, 0, 0',
	X =  158.991  mm,	Y =   -410.760  mm,	Z =   -237.406  mm,
	W =  90.000 deg,	P =   0.000 deg,	R =   90.000 deg
};
P[688]{
   GP1:
	UF : 0, UT : 6,		CONFIG : 'N U T, 0, 0, 0',
	X =  159.626  mm,	Y =   -411.893  mm,	Z =   -237.155  mm,
	W =  90.000 deg,	P =   0.000 deg,	R =   90.000 deg
};
P[689]{
   GP1:
	UF : 0, UT : 6,		CONFIG : 'N U T, 0, 0, 0',
	X =  160.358  mm,	Y =   -413.163  mm,	Z =   -237.143  mm,
	W =  90.000 deg,	P =   0.000 deg,	R =   90.000 deg
};
P[690]{
   GP1:
	UF : 0, UT : 6,		CONFIG : 'N U T, 0, 0, 0',
	X =  160.807  mm,	Y =   -413.895  mm,	Z =   -237.477  mm,
	W =  90.000 deg,	P =   0.000 deg,	R =   90.000 deg
};
P[691]{
   GP1:
	UF : 0, UT : 6,		CONFIG : 'N U T, 0, 0, 0',
	X =  161.217  mm,	Y =   -414.606  mm,	Z =   -237.465  mm,
	W =  90.000 deg,	P =   0.000 deg,	R =   90.000 deg
};
P[692]{
   GP1:
	UF : 0, UT : 6,		CONFIG : 'N U T, 0, 0, 0',
	X =  161.574  mm,	Y =   -415.215  mm,	Z =   -237.534  mm,
	W =  90.000 deg,	P =   0.000 deg,	R =   90.000 deg
};
P[693]{
   GP1:
	UF : 0, UT : 6,		CONFIG : 'N U T, 0, 0, 0',
	X =  162.165  mm,	Y =   -416.293  mm,	Z =   -237.135  mm,
	W =  90.000 deg,	P =   0.000 deg,	R =   90.000 deg
};
P[694]{
   GP1:
	UF : 0, UT : 6,		CONFIG : 'N U T, 0, 0, 0',
	X =  162.450  mm,	Y =   -416.727  mm,	Z =   -237.574  mm,
	W =  90.000 deg,	P =   0.000 deg,	R =   90.000 deg
};
P[695]{
   GP1:
	UF : 0, UT : 6,		CONFIG : 'N U T, 0, 0, 0',
	X =  162.888  mm,	Y =   -417.498  mm,	Z =   -237.478  mm,
	W =  90.000 deg,	P =   0.000 deg,	R =   90.000 deg
};
P[696]{
   GP1:
	UF : 0, UT : 6,		CONFIG : 'N U T, 0, 0, 0',
	X =  163.340  mm,	Y =   -418.331  mm,	Z =   -237.128  mm,
	W =  90.000 deg,	P =   0.000 deg,	R =   90.000 deg
};
P[697]{
   GP1:
	UF : 0, UT : 6,		CONFIG : 'N U T, 0, 0, 0',
	X =  163.683  mm,	Y =   -418.877  mm,	Z =   -237.459  mm,
	W =  90.000 deg,	P =   0.000 deg,	R =   90.000 deg
};
P[698]{
   GP1:
	UF : 0, UT : 6,		CONFIG : 'N U T, 0, 0, 0',
	X =  163.965  mm,	Y =   -419.415  mm,	Z =   -237.113  mm,
	W =  90.000 deg,	P =   0.000 deg,	R =   90.000 deg
};
P[699]{
   GP1:
	UF : 0, UT : 6,		CONFIG : 'N U T, 0, 0, 0',
	X =  164.140  mm,	Y =   -419.661  mm,	Z =   -237.509  mm,
	W =  90.000 deg,	P =   0.000 deg,	R =   90.000 deg
};
P[700]{
   GP1:
	UF : 0, UT : 6,		CONFIG : 'N U T, 0, 0, 0',
	X =  164.569  mm,	Y =   -420.457  mm,	Z =   -237.148  mm,
	W =  90.000 deg,	P =   0.000 deg,	R =   90.000 deg
};
P[701]{
   GP1:
	UF : 0, UT : 6,		CONFIG : 'N U T, 0, 0, 0',
	X =  164.968  mm,	Y =   -421.096  mm,	Z =   -237.501  mm,
	W =  90.000 deg,	P =   0.000 deg,	R =   90.000 deg
};
P[702]{
   GP1:
	UF : 0, UT : 6,		CONFIG : 'N U T, 0, 0, 0',
	X =  165.315  mm,	Y =   -421.655  mm,	Z =   -237.590  mm,
	W =  90.000 deg,	P =   0.000 deg,	R =   90.000 deg
};
P[703]{
   GP1:
	UF : 0, UT : 6,		CONFIG : 'N U T, 0, 0, 0',
	X =  165.888  mm,	Y =   -422.497  mm,	Z =   -237.429  mm,
	W =  90.000 deg,	P =   0.000 deg,	R =   90.000 deg
};
P[704]{
   GP1:
	UF : 0, UT : 6,		CONFIG : 'N U T, 0, 0, 0',
	X =  167.683  mm,	Y =   -424.199  mm,	Z =   -237.468  mm,
	W =  90.000 deg,	P =   0.000 deg,	R =   90.000 deg
};
P[705]{
   GP1:
	UF : 0, UT : 6,		CONFIG : 'N U T, 0, 0, 0',
	X =  168.020  mm,	Y =   -424.396  mm,	Z =   -237.550  mm,
	W =  90.000 deg,	P =   0.000 deg,	R =   90.000 deg
};
P[706]{
   GP1:
	UF : 0, UT : 6,		CONFIG : 'N U T, 0, 0, 0',
	X =  169.785  mm,	Y =   -425.248  mm,	Z =   -237.510  mm,
	W =  90.000 deg,	P =   0.000 deg,	R =   90.000 deg
};
P[707]{
   GP1:
	UF : 0, UT : 6,		CONFIG : 'N U T, 0, 0, 0',
	X =  170.974  mm,	Y =   -425.565  mm,	Z =   -237.444  mm,
	W =  90.000 deg,	P =   0.000 deg,	R =   90.000 deg
};
P[708]{
   GP1:
	UF : 0, UT : 6,		CONFIG : 'N U T, 0, 0, 0',
	X =  172.156  mm,	Y =   -425.697  mm,	Z =   -237.553  mm,
	W =  90.000 deg,	P =   0.000 deg,	R =   90.000 deg
};
P[709]{
   GP1:
	UF : 0, UT : 6,		CONFIG : 'N U T, 0, 0, 0',
	X =  172.924  mm,	Y =   -425.696  mm,	Z =   -237.532  mm,
	W =  90.000 deg,	P =   0.000 deg,	R =   90.000 deg
};
P[710]{
   GP1:
	UF : 0, UT : 6,		CONFIG : 'N U T, 0, 0, 0',
	X =  173.371  mm,	Y =   -425.681  mm,	Z =   -237.525  mm,
	W =  90.000 deg,	P =   0.000 deg,	R =   90.000 deg
};
P[711]{
   GP1:
	UF : 0, UT : 6,		CONFIG : 'N U T, 0, 0, 0',
	X =  173.967  mm,	Y =   -425.580  mm,	Z =   -237.545  mm,
	W =  90.000 deg,	P =   0.000 deg,	R =   90.000 deg
};
P[712]{
   GP1:
	UF : 0, UT : 6,		CONFIG : 'N U T, 0, 0, 0',
	X =  174.875  mm,	Y =   -425.384  mm,	Z =   -237.441  mm,
	W =  90.000 deg,	P =   0.000 deg,	R =   90.000 deg
};
P[713]{
   GP1:
	UF : 0, UT : 6,		CONFIG : 'N U T, 0, 0, 0',
	X =  177.076  mm,	Y =   -424.413  mm,	Z =   -237.545  mm,
	W =  90.000 deg,	P =   0.000 deg,	R =   90.000 deg
};
P[714]{
   GP1:
	UF : 0, UT : 6,		CONFIG : 'N U T, 0, 0, 0',
	X =  177.929  mm,	Y =   -423.919  mm,	Z =   -237.564  mm,
	W =  90.000 deg,	P =   0.000 deg,	R =   90.000 deg
};
P[715]{
   GP1:
	UF : 0, UT : 6,		CONFIG : 'N U T, 0, 0, 0',
	X =  178.620  mm,	Y =   -423.529  mm,	Z =   -237.457  mm,
	W =  90.000 deg,	P =   0.000 deg,	R =   90.000 deg
};
P[716]{
   GP1:
	UF : 0, UT : 6,		CONFIG : 'N U T, 0, 0, 0',
	X =  179.330  mm,	Y =   -423.147  mm,	Z =   -237.115  mm,
	W =  90.000 deg,	P =   0.000 deg,	R =   90.000 deg
};
P[717]{
   GP1:
	UF : 0, UT : 6,		CONFIG : 'N U T, 0, 0, 0',
	X =  180.807  mm,	Y =   -422.263  mm,	Z =   -237.491  mm,
	W =  90.000 deg,	P =   0.000 deg,	R =   90.000 deg
};
P[718]{
   GP1:
	UF : 0, UT : 6,		CONFIG : 'N U T, 0, 0, 0',
	X =  183.007  mm,	Y =   -420.991  mm,	Z =   -237.516  mm,
	W =  90.000 deg,	P =   0.000 deg,	R =   90.000 deg
};
P[719]{
   GP1:
	UF : 0, UT : 6,		CONFIG : 'N U T, 0, 0, 0',
	X =  183.564  mm,	Y =   -420.704  mm,	Z =   -237.092  mm,
	W =  90.000 deg,	P =   0.000 deg,	R =   90.000 deg
};
P[720]{
   GP1:
	UF : 0, UT : 6,		CONFIG : 'N U T, 0, 0, 0',
	X =  183.770  mm,	Y =   -420.546  mm,	Z =   -237.576  mm,
	W =  90.000 deg,	P =   0.000 deg,	R =   90.000 deg
};
P[721]{
   GP1:
	UF : 0, UT : 6,		CONFIG : 'N U T, 0, 0, 0',
	X =  184.668  mm,	Y =   -420.065  mm,	Z =   -237.108  mm,
	W =  90.000 deg,	P =   0.000 deg,	R =   90.000 deg
};
P[722]{
   GP1:
	UF : 0, UT : 6,		CONFIG : 'N U T, 0, 0, 0',
	X =  186.687  mm,	Y =   -418.871  mm,	Z =   -237.465  mm,
	W =  90.000 deg,	P =   0.000 deg,	R =   90.000 deg
};
P[723]{
   GP1:
	UF : 0, UT : 6,		CONFIG : 'N U T, 0, 0, 0',
	X =  188.917  mm,	Y =   -417.578  mm,	Z =   -237.520  mm,
	W =  90.000 deg,	P =   0.000 deg,	R =   90.000 deg
};
P[724]{
   GP1:
	UF : 0, UT : 6,		CONFIG : 'N U T, 0, 0, 0',
	X =  189.688  mm,	Y =   -417.168  mm,	Z =   -237.092  mm,
	W =  90.000 deg,	P =   0.000 deg,	R =   90.000 deg
};
P[725]{
   GP1:
	UF : 0, UT : 6,		CONFIG : 'N U T, 0, 0, 0',
	X =  190.296  mm,	Y =   -416.816  mm,	Z =   -237.094  mm,
	W =  90.000 deg,	P =   0.000 deg,	R =   90.000 deg
};
P[726]{
   GP1:
	UF : 0, UT : 6,		CONFIG : 'N U T, 0, 0, 0',
	X =  190.516  mm,	Y =   -416.657  mm,	Z =   -237.498  mm,
	W =  90.000 deg,	P =   0.000 deg,	R =   90.000 deg
};
P[727]{
   GP1:
	UF : 0, UT : 6,		CONFIG : 'N U T, 0, 0, 0',
	X =  192.480  mm,	Y =   -415.521  mm,	Z =   -237.524  mm,
	W =  90.000 deg,	P =   0.000 deg,	R =   90.000 deg
};
P[728]{
   GP1:
	UF : 0, UT : 6,		CONFIG : 'N U T, 0, 0, 0',
	X =  193.357  mm,	Y =   -415.013  mm,	Z =   -237.532  mm,
	W =  90.000 deg,	P =   0.000 deg,	R =   90.000 deg
};
P[729]{
   GP1:
	UF : 0, UT : 6,		CONFIG : 'N U T, 0, 0, 0',
	X =  194.903  mm,	Y =   -414.153  mm,	Z =   -237.133  mm,
	W =  90.000 deg,	P =   0.000 deg,	R =   90.000 deg
};
P[730]{
   GP1:
	UF : 0, UT : 6,		CONFIG : 'N U T, 0, 0, 0',
	X =  195.633  mm,	Y =   -413.699  mm,	Z =   -237.544  mm,
	W =  90.000 deg,	P =   0.000 deg,	R =   90.000 deg
};
P[731]{
   GP1:
	UF : 0, UT : 6,		CONFIG : 'N U T, 0, 0, 0',
	X =  196.990  mm,	Y =   -412.914  mm,	Z =   -237.563  mm,
	W =  90.000 deg,	P =   0.000 deg,	R =   90.000 deg
};
P[732]{
   GP1:
	UF : 0, UT : 6,		CONFIG : 'N U T, 0, 0, 0',
	X =  197.414  mm,	Y =   -412.702  mm,	Z =   -237.151  mm,
	W =  90.000 deg,	P =   0.000 deg,	R =   90.000 deg
};
P[733]{
   GP1:
	UF : 0, UT : 6,		CONFIG : 'N U T, 0, 0, 0',
	X =  198.524  mm,	Y =   -412.029  mm,	Z =   -237.555  mm,
	W =  90.000 deg,	P =   0.000 deg,	R =   90.000 deg
};
P[734]{
   GP1:
	UF : 0, UT : 6,		CONFIG : 'N U T, 0, 0, 0',
	X =  199.140  mm,	Y =   -411.673  mm,	Z =   -237.553  mm,
	W =  90.000 deg,	P =   0.000 deg,	R =   90.000 deg
};
P[735]{
   GP1:
	UF : 0, UT : 6,		CONFIG : 'N U T, 0, 0, 0',
	X =  199.923  mm,	Y =   -411.218  mm,	Z =   -237.588  mm,
	W =  90.000 deg,	P =   0.000 deg,	R =   90.000 deg
};
P[736]{
   GP1:
	UF : 0, UT : 6,		CONFIG : 'N U T, 0, 0, 0',
	X =  200.600  mm,	Y =   -410.862  mm,	Z =   -237.158  mm,
	W =  90.000 deg,	P =   0.000 deg,	R =   90.000 deg
};
P[737]{
   GP1:
	UF : 0, UT : 6,		CONFIG : 'N U T, 0, 0, 0',
	X =  201.446  mm,	Y =   -410.342  mm,	Z =   -237.543  mm,
	W =  90.000 deg,	P =   0.000 deg,	R =   90.000 deg
};
P[738]{
   GP1:
	UF : 0, UT : 6,		CONFIG : 'N U T, 0, 0, 0',
	X =  202.079  mm,	Y =   -410.010  mm,	Z =   -237.133  mm,
	W =  90.000 deg,	P =   0.000 deg,	R =   90.000 deg
};
P[739]{
   GP1:
	UF : 0, UT : 6,		CONFIG : 'N U T, 0, 0, 0',
	X =  204.362  mm,	Y =   -408.691  mm,	Z =   -237.153  mm,
	W =  90.000 deg,	P =   0.000 deg,	R =   90.000 deg
};
P[740]{
   GP1:
	UF : 0, UT : 6,		CONFIG : 'N U T, 0, 0, 0',
	X =  204.402  mm,	Y =   -408.639  mm,	Z =   -237.501  mm,
	W =  90.000 deg,	P =   0.000 deg,	R =   90.000 deg
};
P[741]{
   GP1:
	UF : 0, UT : 6,		CONFIG : 'N U T, 0, 0, 0',
	X =  205.130  mm,	Y =   -408.216  mm,	Z =   -237.532  mm,
	W =  90.000 deg,	P =   0.000 deg,	R =   90.000 deg
};
P[742]{
   GP1:
	UF : 0, UT : 6,		CONFIG : 'N U T, 0, 0, 0',
	X =  205.769  mm,	Y =   -407.882  mm,	Z =   -237.096  mm,
	W =  90.000 deg,	P =   0.000 deg,	R =   90.000 deg
};
P[743]{
   GP1:
	UF : 0, UT : 6,		CONFIG : 'N U T, 0, 0, 0',
	X =  206.636  mm,	Y =   -407.342  mm,	Z =   -237.580  mm,
	W =  90.000 deg,	P =   0.000 deg,	R =   90.000 deg
};
P[744]{
   GP1:
	UF : 0, UT : 6,		CONFIG : 'N U T, 0, 0, 0',
	X =  207.259  mm,	Y =   -407.002  mm,	Z =   -237.346  mm,
	W =  90.000 deg,	P =   0.000 deg,	R =   90.000 deg
};
P[745]{
   GP1:
	UF : 0, UT : 6,		CONFIG : 'N U T, 0, 0, 0',
	X =  208.289  mm,	Y =   -406.425  mm,	Z =   -237.125  mm,
	W =  90.000 deg,	P =   0.000 deg,	R =   90.000 deg
};
P[746]{
   GP1:
	UF : 0, UT : 6,		CONFIG : 'N U T, 0, 0, 0',
	X =  208.552  mm,	Y =   -406.273  mm,	Z =   -237.123  mm,
	W =  90.000 deg,	P =   0.000 deg,	R =   90.000 deg
};
P[747]{
   GP1:
	UF : 0, UT : 6,		CONFIG : 'N U T, 0, 0, 0',
	X =  209.569  mm,	Y =   -405.652  mm,	Z =   -237.554  mm,
	W =  90.000 deg,	P =   0.000 deg,	R =   90.000 deg
};
P[748]{
   GP1:
	UF : 0, UT : 6,		CONFIG : 'N U T, 0, 0, 0',
	X =  210.924  mm,	Y =   -404.873  mm,	Z =   -237.512  mm,
	W =  90.000 deg,	P =   0.000 deg,	R =   90.000 deg
};
P[749]{
   GP1:
	UF : 0, UT : 6,		CONFIG : 'N U T, 0, 0, 0',
	X =  211.599  mm,	Y =   -404.511  mm,	Z =   -237.157  mm,
	W =  90.000 deg,	P =   0.000 deg,	R =   90.000 deg
};
P[750]{
   GP1:
	UF : 0, UT : 6,		CONFIG : 'N U T, 0, 0, 0',
	X =  212.426  mm,	Y =   -404.006  mm,	Z =   -237.498  mm,
	W =  90.000 deg,	P =   0.000 deg,	R =   90.000 deg
};
P[751]{
   GP1:
	UF : 0, UT : 6,		CONFIG : 'N U T, 0, 0, 0',
	X =  213.964  mm,	Y =   -403.114  mm,	Z =   -237.552  mm,
	W =  90.000 deg,	P =   0.000 deg,	R =   90.000 deg
};
P[752]{
   GP1:
	UF : 0, UT : 6,		CONFIG : 'N U T, 0, 0, 0',
	X =  213.972  mm,	Y =   -403.146  mm,	Z =   -237.104  mm,
	W =  90.000 deg,	P =   0.000 deg,	R =   90.000 deg
};
P[753]{
   GP1:
	UF : 0, UT : 6,		CONFIG : 'N U T, 0, 0, 0',
	X =  214.593  mm,	Y =   -402.784  mm,	Z =   -237.148  mm,
	W =  90.000 deg,	P =   0.000 deg,	R =   90.000 deg
};
P[754]{
   GP1:
	UF : 0, UT : 6,		CONFIG : 'N U T, 0, 0, 0',
	X =  215.120  mm,	Y =   -402.482  mm,	Z =   -237.117  mm,
	W =  90.000 deg,	P =   0.000 deg,	R =   90.000 deg
};
P[755]{
   GP1:
	UF : 0, UT : 6,		CONFIG : 'N U T, 0, 0, 0',
	X =  215.520  mm,	Y =   -402.219  mm,	Z =   -237.509  mm,
	W =  90.000 deg,	P =   0.000 deg,	R =   90.000 deg
};
P[756]{
   GP1:
	UF : 0, UT : 6,		CONFIG : 'N U T, 0, 0, 0',
	X =  216.873  mm,	Y =   -401.438  mm,	Z =   -237.507  mm,
	W =  90.000 deg,	P =   0.000 deg,	R =   90.000 deg
};
P[757]{
   GP1:
	UF : 0, UT : 6,		CONFIG : 'N U T, 0, 0, 0',
	X =  217.110  mm,	Y =   -401.334  mm,	Z =   -237.096  mm,
	W =  90.000 deg,	P =   0.000 deg,	R =   90.000 deg
};
P[758]{
   GP1:
	UF : 0, UT : 6,		CONFIG : 'N U T, 0, 0, 0',
	X =  217.981  mm,	Y =   -400.826  mm,	Z =   -237.155  mm,
	W =  90.000 deg,	P =   0.000 deg,	R =   90.000 deg
};
P[759]{
   GP1:
	UF : 0, UT : 6,		CONFIG : 'N U T, 0, 0, 0',
	X =  218.260  mm,	Y =   -400.669  mm,	Z =   -237.114  mm,
	W =  90.000 deg,	P =   0.000 deg,	R =   90.000 deg
};
P[760]{
   GP1:
	UF : 0, UT : 6,		CONFIG : 'N U T, 0, 0, 0',
	X =  219.100  mm,	Y =   -400.150  mm,	Z =   -237.531  mm,
	W =  90.000 deg,	P =   0.000 deg,	R =   90.000 deg
};
P[761]{
   GP1:
	UF : 0, UT : 6,		CONFIG : 'N U T, 0, 0, 0',
	X =  219.581  mm,	Y =   -399.903  mm,	Z =   -237.147  mm,
	W =  90.000 deg,	P =   0.000 deg,	R =   90.000 deg
};
P[762]{
   GP1:
	UF : 0, UT : 6,		CONFIG : 'N U T, 0, 0, 0',
	X =  219.917  mm,	Y =   -399.674  mm,	Z =   -237.590  mm,
	W =  90.000 deg,	P =   0.000 deg,	R =   90.000 deg
};
P[763]{
   GP1:
	UF : 0, UT : 6,		CONFIG : 'N U T, 0, 0, 0',
	X =  220.617  mm,	Y =   -399.277  mm,	Z =   -237.486  mm,
	W =  90.000 deg,	P =   0.000 deg,	R =   90.000 deg
};
P[764]{
   GP1:
	UF : 0, UT : 6,		CONFIG : 'N U T, 0, 0, 0',
	X =  223.515  mm,	Y =   -397.596  mm,	Z =   -237.588  mm,
	W =  90.000 deg,	P =   0.000 deg,	R =   90.000 deg
};
P[765]{
   GP1:
	UF : 0, UT : 6,		CONFIG : 'N U T, 0, 0, 0',
	X =  224.279  mm,	Y =   -397.158  mm,	Z =   -237.545  mm,
	W =  90.000 deg,	P =   0.000 deg,	R =   90.000 deg
};
P[766]{
   GP1:
	UF : 0, UT : 6,		CONFIG : 'N U T, 0, 0, 0',
	X =  225.153  mm,	Y =   -396.687  mm,	Z =   -237.134  mm,
	W =  90.000 deg,	P =   0.000 deg,	R =   90.000 deg
};
P[767]{
   GP1:
	UF : 0, UT : 6,		CONFIG : 'N U T, 0, 0, 0',
	X =  225.427  mm,	Y =   -396.529  mm,	Z =   -237.132  mm,
	W =  90.000 deg,	P =   0.000 deg,	R =   90.000 deg
};
P[768]{
   GP1:
	UF : 0, UT : 6,		CONFIG : 'N U T, 0, 0, 0',
	X =  226.333  mm,	Y =   -396.005  mm,	Z =   -237.143  mm,
	W =  90.000 deg,	P =   0.000 deg,	R =   90.000 deg
};
P[769]{
   GP1:
	UF : 0, UT : 6,		CONFIG : 'N U T, 0, 0, 0',
	X =  227.551  mm,	Y =   -395.302  mm,	Z =   -237.136  mm,
	W =  90.000 deg,	P =   0.000 deg,	R =   90.000 deg
};
P[770]{
   GP1:
	UF : 0, UT : 6,		CONFIG : 'N U T, 0, 0, 0',
	X =  228.006  mm,	Y =   -395.012  mm,	Z =   -237.478  mm,
	W =  90.000 deg,	P =   0.000 deg,	R =   90.000 deg
};
P[771]{
   GP1:
	UF : 0, UT : 6,		CONFIG : 'N U T, 0, 0, 0',
	X =  228.600  mm,	Y =   -394.698  mm,	Z =   -237.122  mm,
	W =  90.000 deg,	P =   0.000 deg,	R =   90.000 deg
};
P[772]{
   GP1:
	UF : 0, UT : 6,		CONFIG : 'N U T, 0, 0, 0',
	X =  229.415  mm,	Y =   -394.197  mm,	Z =   -237.499  mm,
	W =  90.000 deg,	P =   0.000 deg,	R =   90.000 deg
};
P[773]{
   GP1:
	UF : 0, UT : 6,		CONFIG : 'N U T, 0, 0, 0',
	X =  230.139  mm,	Y =   -393.774  mm,	Z =   -237.565  mm,
	W =  90.000 deg,	P =   0.000 deg,	R =   90.000 deg
};
P[774]{
   GP1:
	UF : 0, UT : 6,		CONFIG : 'N U T, 0, 0, 0',
	X =  230.218  mm,	Y =   -393.764  mm,	Z =   -237.118  mm,
	W =  90.000 deg,	P =   0.000 deg,	R =   90.000 deg
};
P[775]{
   GP1:
	UF : 0, UT : 6,		CONFIG : 'N U T, 0, 0, 0',
	X =  230.956  mm,	Y =   -393.307  mm,	Z =   -237.504  mm,
	W =  90.000 deg,	P =   0.000 deg,	R =   90.000 deg
};
P[776]{
   GP1:
	UF : 0, UT : 6,		CONFIG : 'N U T, 0, 0, 0',
	X =  232.421  mm,	Y =   -392.464  mm,	Z =   -237.462  mm,
	W =  90.000 deg,	P =   0.000 deg,	R =   90.000 deg
};
P[777]{
   GP1:
	UF : 0, UT : 6,		CONFIG : 'N U T, 0, 0, 0',
	X =  233.245  mm,	Y =   -391.978  mm,	Z =   -237.584  mm,
	W =  90.000 deg,	P =   0.000 deg,	R =   90.000 deg
};
P[778]{
   GP1:
	UF : 0, UT : 6,		CONFIG : 'N U T, 0, 0, 0',
	X =  233.655  mm,	Y =   -391.776  mm,	Z =   -237.158  mm,
	W =  90.000 deg,	P =   0.000 deg,	R =   90.000 deg
};
P[779]{
   GP1:
	UF : 0, UT : 6,		CONFIG : 'N U T, 0, 0, 0',
	X =  234.487  mm,	Y =   -391.268  mm,	Z =   -237.503  mm,
	W =  90.000 deg,	P =   0.000 deg,	R =   90.000 deg
};
P[780]{
   GP1:
	UF : 0, UT : 6,		CONFIG : 'N U T, 0, 0, 0',
	X =  235.250  mm,	Y =   -390.822  mm,	Z =   -237.573  mm,
	W =  90.000 deg,	P =   0.000 deg,	R =   90.000 deg
};
P[781]{
   GP1:
	UF : 0, UT : 6,		CONFIG : 'N U T, 0, 0, 0',
	X =  236.107  mm,	Y =   -390.330  mm,	Z =   -237.545  mm,
	W =  90.000 deg,	P =   0.000 deg,	R =   90.000 deg
};
P[782]{
   GP1:
	UF : 0, UT : 6,		CONFIG : 'N U T, 0, 0, 0',
	X =  236.799  mm,	Y =   -389.934  mm,	Z =   -237.494  mm,
	W =  90.000 deg,	P =   0.000 deg,	R =   90.000 deg
};
P[783]{
   GP1:
	UF : 0, UT : 6,		CONFIG : 'N U T, 0, 0, 0',
	X =  237.438  mm,	Y =   -389.571  mm,	Z =   -237.414  mm,
	W =  90.000 deg,	P =   0.000 deg,	R =   90.000 deg
};
P[784]{
   GP1:
	UF : 0, UT : 6,		CONFIG : 'N U T, 0, 0, 0',
	X =  238.366  mm,	Y =   -389.060  mm,	Z =   -237.116  mm,
	W =  90.000 deg,	P =   0.000 deg,	R =   90.000 deg
};
P[785]{
   GP1:
	UF : 0, UT : 6,		CONFIG : 'N U T, 0, 0, 0',
	X =  240.055  mm,	Y =   -388.083  mm,	Z =   -237.119  mm,
	W =  90.000 deg,	P =   0.000 deg,	R =   90.000 deg
};
P[786]{
   GP1:
	UF : 0, UT : 6,		CONFIG : 'N U T, 0, 0, 0',
	X =  240.526  mm,	Y =   -387.780  mm,	Z =   -237.520  mm,
	W =  90.000 deg,	P =   0.000 deg,	R =   90.000 deg
};
P[787]{
   GP1:
	UF : 0, UT : 6,		CONFIG : 'N U T, 0, 0, 0',
	X =  241.124  mm,	Y =   -387.429  mm,	Z =   -237.591  mm,
	W =  90.000 deg,	P =   0.000 deg,	R =   90.000 deg
};
P[788]{
   GP1:
	UF : 0, UT : 6,		CONFIG : 'N U T, 0, 0, 0',
	X =  241.536  mm,	Y =   -387.228  mm,	Z =   -237.127  mm,
	W =  90.000 deg,	P =   0.000 deg,	R =   90.000 deg
};
P[789]{
   GP1:
	UF : 0, UT : 6,		CONFIG : 'N U T, 0, 0, 0',
	X =  242.397  mm,	Y =   -386.733  mm,	Z =   -237.096  mm,
	W =  90.000 deg,	P =   0.000 deg,	R =   90.000 deg
};
P[790]{
   GP1:
	UF : 0, UT : 6,		CONFIG : 'N U T, 0, 0, 0',
	X =  242.772  mm,	Y =   -386.483  mm,	Z =   -237.515  mm,
	W =  90.000 deg,	P =   0.000 deg,	R =   90.000 deg
};
P[791]{
   GP1:
	UF : 0, UT : 6,		CONFIG : 'N U T, 0, 0, 0',
	X =  243.451  mm,	Y =   -386.089  mm,	Z =   -237.545  mm,
	W =  90.000 deg,	P =   0.000 deg,	R =   90.000 deg
};
P[792]{
   GP1:
	UF : 0, UT : 6,		CONFIG : 'N U T, 0, 0, 0',
	X =  244.942  mm,	Y =   -385.228  mm,	Z =   -237.550  mm,
	W =  90.000 deg,	P =   0.000 deg,	R =   90.000 deg
};
P[793]{
   GP1:
	UF : 0, UT : 6,		CONFIG : 'N U T, 0, 0, 0',
	X =  245.613  mm,	Y =   -384.846  mm,	Z =   -237.471  mm,
	W =  90.000 deg,	P =   0.000 deg,	R =   90.000 deg
};
P[794]{
   GP1:
	UF : 0, UT : 6,		CONFIG : 'N U T, 0, 0, 0',
	X =  246.227  mm,	Y =   -384.485  mm,	Z =   -237.565  mm,
	W =  90.000 deg,	P =   0.000 deg,	R =   90.000 deg
};
P[795]{
   GP1:
	UF : 0, UT : 6,		CONFIG : 'N U T, 0, 0, 0',
	X =  247.907  mm,	Y =   -383.515  mm,	Z =   -237.553  mm,
	W =  90.000 deg,	P =   0.000 deg,	R =   90.000 deg
};
P[796]{
   GP1:
	UF : 0, UT : 6,		CONFIG : 'N U T, 0, 0, 0',
	X =  248.024  mm,	Y =   -383.482  mm,	Z =   -237.131  mm,
	W =  90.000 deg,	P =   0.000 deg,	R =   90.000 deg
};
P[797]{
   GP1:
	UF : 0, UT : 6,		CONFIG : 'N U T, 0, 0, 0',
	X =  248.565  mm,	Y =   -383.138  mm,	Z =   -237.515  mm,
	W =  90.000 deg,	P =   0.000 deg,	R =   90.000 deg
};
P[798]{
   GP1:
	UF : 0, UT : 6,		CONFIG : 'N U T, 0, 0, 0',
	X =  249.285  mm,	Y =   -382.723  mm,	Z =   -237.506  mm,
	W =  90.000 deg,	P =   0.000 deg,	R =   90.000 deg
};
P[799]{
   GP1:
	UF : 0, UT : 6,		CONFIG : 'N U T, 0, 0, 0',
	X =  249.899  mm,	Y =   -382.400  mm,	Z =   -237.121  mm,
	W =  90.000 deg,	P =   0.000 deg,	R =   90.000 deg
};
P[800]{
   GP1:
	UF : 0, UT : 6,		CONFIG : 'N U T, 0, 0, 0',
	X =  250.698  mm,	Y =   -381.907  mm,	Z =   -237.512  mm,
	W =  90.000 deg,	P =   0.000 deg,	R =   90.000 deg
};
P[801]{
   GP1:
	UF : 0, UT : 6,		CONFIG : 'N U T, 0, 0, 0',
	X =  251.537  mm,	Y =   -381.417  mm,	Z =   -237.579  mm,
	W =  90.000 deg,	P =   0.000 deg,	R =   90.000 deg
};
P[802]{
   GP1:
	UF : 0, UT : 6,		CONFIG : 'N U T, 0, 0, 0',
	X =  252.223  mm,	Y =   -381.024  mm,	Z =   -237.548  mm,
	W =  90.000 deg,	P =   0.000 deg,	R =   90.000 deg
};
P[803]{
   GP1:
	UF : 0, UT : 6,		CONFIG : 'N U T, 0, 0, 0',
	X =  252.895  mm,	Y =   -380.637  mm,	Z =   -237.531  mm,
	W =  90.000 deg,	P =   0.000 deg,	R =   90.000 deg
};
P[804]{
   GP1:
	UF : 0, UT : 6,		CONFIG : 'N U T, 0, 0, 0',
	X =  253.696  mm,	Y =   -380.176  mm,	Z =   -237.507  mm,
	W =  90.000 deg,	P =   0.000 deg,	R =   90.000 deg
};
P[805]{
   GP1:
	UF : 0, UT : 6,		CONFIG : 'N U T, 0, 0, 0',
	X =  255.150  mm,	Y =   -379.340  mm,	Z =   -237.466  mm,
	W =  90.000 deg,	P =   0.000 deg,	R =   90.000 deg
};
P[806]{
   GP1:
	UF : 0, UT : 6,		CONFIG : 'N U T, 0, 0, 0',
	X =  256.559  mm,	Y =   -378.519  mm,	Z =   -237.563  mm,
	W =  90.000 deg,	P =   0.000 deg,	R =   90.000 deg
};
P[807]{
   GP1:
	UF : 0, UT : 6,		CONFIG : 'N U T, 0, 0, 0',
	X =  256.658  mm,	Y =   -378.499  mm,	Z =   -237.095  mm,
	W =  90.000 deg,	P =   0.000 deg,	R =   90.000 deg
};
P[808]{
   GP1:
	UF : 0, UT : 6,		CONFIG : 'N U T, 0, 0, 0',
	X =  258.495  mm,	Y =   -377.435  mm,	Z =   -237.148  mm,
	W =  90.000 deg,	P =   0.000 deg,	R =   90.000 deg
};
P[809]{
   GP1:
	UF : 0, UT : 6,		CONFIG : 'N U T, 0, 0, 0',
	X =  259.248  mm,	Y =   -376.999  mm,	Z =   -237.157  mm,
	W =  90.000 deg,	P =   0.000 deg,	R =   90.000 deg
};
P[810]{
   GP1:
	UF : 0, UT : 6,		CONFIG : 'N U T, 0, 0, 0',
	X =  261.072  mm,	Y =   -375.915  mm,	Z =   -237.542  mm,
	W =  90.000 deg,	P =   0.000 deg,	R =   90.000 deg
};
P[811]{
   GP1:
	UF : 0, UT : 6,		CONFIG : 'N U T, 0, 0, 0',
	X =  261.886  mm,	Y =   -375.448  mm,	Z =   -237.498  mm,
	W =  90.000 deg,	P =   0.000 deg,	R =   90.000 deg
};
P[812]{
   GP1:
	UF : 0, UT : 6,		CONFIG : 'N U T, 0, 0, 0',
	X =  262.567  mm,	Y =   -375.051  mm,	Z =   -237.547  mm,
	W =  90.000 deg,	P =   0.000 deg,	R =   90.000 deg
};
P[813]{
   GP1:
	UF : 0, UT : 6,		CONFIG : 'N U T, 0, 0, 0',
	X =  262.629  mm,	Y =   -375.050  mm,	Z =   -237.120  mm,
	W =  90.000 deg,	P =   0.000 deg,	R =   90.000 deg
};
P[814]{
   GP1:
	UF : 0, UT : 6,		CONFIG : 'N U T, 0, 0, 0',
	X =  264.288  mm,	Y =   -374.093  mm,	Z =   -237.107  mm,
	W =  90.000 deg,	P =   0.000 deg,	R =   90.000 deg
};
P[815]{
   GP1:
	UF : 0, UT : 6,		CONFIG : 'N U T, 0, 0, 0',
	X =  264.847  mm,	Y =   -373.735  mm,	Z =   -237.554  mm,
	W =  90.000 deg,	P =   0.000 deg,	R =   90.000 deg
};
P[816]{
   GP1:
	UF : 0, UT : 6,		CONFIG : 'N U T, 0, 0, 0',
	X =  265.626  mm,	Y =   -373.319  mm,	Z =   -237.120  mm,
	W =  90.000 deg,	P =   0.000 deg,	R =   90.000 deg
};
P[817]{
   GP1:
	UF : 0, UT : 6,		CONFIG : 'N U T, 0, 0, 0',
	X =  266.203  mm,	Y =   -372.955  mm,	Z =   -237.507  mm,
	W =  90.000 deg,	P =   0.000 deg,	R =   90.000 deg
};
P[818]{
   GP1:
	UF : 0, UT : 6,		CONFIG : 'N U T, 0, 0, 0',
	X =  266.959  mm,	Y =   -372.549  mm,	Z =   -237.130  mm,
	W =  90.000 deg,	P =   0.000 deg,	R =   90.000 deg
};
P[819]{
   GP1:
	UF : 0, UT : 6,		CONFIG : 'N U T, 0, 0, 0',
	X =  268.428  mm,	Y =   -371.700  mm,	Z =   -237.148  mm,
	W =  90.000 deg,	P =   0.000 deg,	R =   90.000 deg
};
P[820]{
   GP1:
	UF : 0, UT : 6,		CONFIG : 'N U T, 0, 0, 0',
	X =  269.997  mm,	Y =   -370.723  mm,	Z =   -237.482  mm,
	W =  90.000 deg,	P =   0.000 deg,	R =   90.000 deg
};
P[821]{
   GP1:
	UF : 0, UT : 6,		CONFIG : 'N U T, 0, 0, 0',
	X =  270.733  mm,	Y =   -370.177  mm,	Z =   -237.535  mm,
	W =  90.000 deg,	P =   0.000 deg,	R =   90.000 deg
};
P[822]{
   GP1:
	UF : 0, UT : 6,		CONFIG : 'N U T, 0, 0, 0',
	X =  271.349  mm,	Y =   -369.608  mm,	Z =   -237.551  mm,
	W =  90.000 deg,	P =   0.000 deg,	R =   90.000 deg
};
P[823]{
   GP1:
	UF : 0, UT : 6,		CONFIG : 'N U T, 0, 0, 0',
	X =  271.886  mm,	Y =   -368.998  mm,	Z =   -237.553  mm,
	W =  90.000 deg,	P =   0.000 deg,	R =   90.000 deg
};
P[824]{
   GP1:
	UF : 0, UT : 6,		CONFIG : 'N U T, 0, 0, 0',
	X =  272.167  mm,	Y =   -368.664  mm,	Z =   -237.514  mm,
	W =  90.000 deg,	P =   0.000 deg,	R =   90.000 deg
};
P[825]{
   GP1:
	UF : 0, UT : 6,		CONFIG : 'N U T, 0, 0, 0',
	X =  272.492  mm,	Y =   -368.159  mm,	Z =   -237.499  mm,
	W =  90.000 deg,	P =   0.000 deg,	R =   90.000 deg
};
P[826]{
   GP1:
	UF : 0, UT : 6,		CONFIG : 'N U T, 0, 0, 0',
	X =  273.508  mm,	Y =   -365.871  mm,	Z =   -237.313  mm,
	W =  90.000 deg,	P =   0.000 deg,	R =   90.000 deg
};
P[827]{
   GP1:
	UF : 0, UT : 6,		CONFIG : 'N U T, 0, 0, 0',
	X =  273.757  mm,	Y =   -364.180  mm,	Z =   -237.590  mm,
	W =  90.000 deg,	P =   0.000 deg,	R =   90.000 deg
};
P[828]{
   GP1:
	UF : 0, UT : 6,		CONFIG : 'N U T, 0, 0, 0',
	X =  273.667  mm,	Y =   -362.348  mm,	Z =   -237.556  mm,
	W =  90.000 deg,	P =   0.000 deg,	R =   90.000 deg
};
P[829]{
   GP1:
	UF : 0, UT : 6,		CONFIG : 'N U T, 0, 0, 0',
	X =  272.450  mm,	Y =   -359.069  mm,	Z =   -237.500  mm,
	W =  90.000 deg,	P =   0.000 deg,	R =   90.000 deg
};
P[830]{
   GP1:
	UF : 0, UT : 6,		CONFIG : 'N U T, 0, 0, 0',
	X =  272.239  mm,	Y =   -358.649  mm,	Z =   -237.107  mm,
	W =  90.000 deg,	P =   0.000 deg,	R =   90.000 deg
};
P[831]{
   GP1:
	UF : 0, UT : 6,		CONFIG : 'N U T, 0, 0, 0',
	X =  271.172  mm,	Y =   -356.857  mm,	Z =   -237.510  mm,
	W =  90.000 deg,	P =   0.000 deg,	R =   90.000 deg
};
P[832]{
   GP1:
	UF : 0, UT : 6,		CONFIG : 'N U T, 0, 0, 0',
	X =  270.783  mm,	Y =   -356.126  mm,	Z =   -237.099  mm,
	W =  90.000 deg,	P =   0.000 deg,	R =   90.000 deg
};
P[833]{
   GP1:
	UF : 0, UT : 6,		CONFIG : 'N U T, 0, 0, 0',
	X =  269.911  mm,	Y =   -354.677  mm,	Z =   -237.540  mm,
	W =  90.000 deg,	P =   0.000 deg,	R =   90.000 deg
};
P[834]{
   GP1:
	UF : 0, UT : 6,		CONFIG : 'N U T, 0, 0, 0',
	X =  268.692  mm,	Y =   -352.553  mm,	Z =   -237.445  mm,
	W =  90.000 deg,	P =   0.000 deg,	R =   90.000 deg
};
P[835]{
   GP1:
	UF : 0, UT : 6,		CONFIG : 'N U T, 0, 0, 0',
	X =  268.143  mm,	Y =   -351.560  mm,	Z =   -237.142  mm,
	W =  90.000 deg,	P =   0.000 deg,	R =   90.000 deg
};
P[836]{
   GP1:
	UF : 0, UT : 6,		CONFIG : 'N U T, 0, 0, 0',
	X =  267.377  mm,	Y =   -350.293  mm,	Z =   -237.571  mm,
	W =  90.000 deg,	P =   0.000 deg,	R =   90.000 deg
};
P[837]{
   GP1:
	UF : 0, UT : 6,		CONFIG : 'N U T, 0, 0, 0',
	X =  266.932  mm,	Y =   -349.515  mm,	Z =   -237.515  mm,
	W =  90.000 deg,	P =   0.000 deg,	R =   90.000 deg
};
P[838]{
   GP1:
	UF : 0, UT : 6,		CONFIG : 'N U T, 0, 0, 0',
	X =  266.120  mm,	Y =   -348.116  mm,	Z =   -237.568  mm,
	W =  90.000 deg,	P =   0.000 deg,	R =   90.000 deg
};
P[839]{
   GP1:
	UF : 0, UT : 6,		CONFIG : 'N U T, 0, 0, 0',
	X =  265.604  mm,	Y =   -347.216  mm,	Z =   -237.521  mm,
	W =  90.000 deg,	P =   0.000 deg,	R =   90.000 deg
};
P[840]{
   GP1:
	UF : 0, UT : 6,		CONFIG : 'N U T, 0, 0, 0',
	X =  265.129  mm,	Y =   -346.339  mm,	Z =   -237.136  mm,
	W =  90.000 deg,	P =   0.000 deg,	R =   90.000 deg
};
P[841]{
   GP1:
	UF : 0, UT : 6,		CONFIG : 'N U T, 0, 0, 0',
	X =  264.866  mm,	Y =   -345.881  mm,	Z =   -237.118  mm,
	W =  90.000 deg,	P =   0.000 deg,	R =   90.000 deg
};
P[842]{
   GP1:
	UF : 0, UT : 6,		CONFIG : 'N U T, 0, 0, 0',
	X =  264.372  mm,	Y =   -345.083  mm,	Z =   -237.530  mm,
	W =  90.000 deg,	P =   0.000 deg,	R =   90.000 deg
};
P[843]{
   GP1:
	UF : 0, UT : 6,		CONFIG : 'N U T, 0, 0, 0',
	X =  264.372  mm,	Y =   -345.020  mm,	Z =   -237.092  mm,
	W =  90.000 deg,	P =   0.000 deg,	R =   90.000 deg
};
P[844]{
   GP1:
	UF : 0, UT : 6,		CONFIG : 'N U T, 0, 0, 0',
	X =  263.540  mm,	Y =   -343.637  mm,	Z =   -237.496  mm,
	W =  90.000 deg,	P =   0.000 deg,	R =   90.000 deg
};
P[845]{
   GP1:
	UF : 0, UT : 6,		CONFIG : 'N U T, 0, 0, 0',
	X =  263.546  mm,	Y =   -343.592  mm,	Z =   -237.103  mm,
	W =  90.000 deg,	P =   0.000 deg,	R =   90.000 deg
};
P[846]{
   GP1:
	UF : 0, UT : 6,		CONFIG : 'N U T, 0, 0, 0',
	X =  262.742  mm,	Y =   -342.263  mm,	Z =   -237.555  mm,
	W =  90.000 deg,	P =   0.000 deg,	R =   90.000 deg
};
P[847]{
   GP1:
	UF : 0, UT : 6,		CONFIG : 'N U T, 0, 0, 0',
	X =  262.294  mm,	Y =   -341.490  mm,	Z =   -237.573  mm,
	W =  90.000 deg,	P =   0.000 deg,	R =   90.000 deg
};
P[848]{
   GP1:
	UF : 0, UT : 6,		CONFIG : 'N U T, 0, 0, 0',
	X =  262.172  mm,	Y =   -341.217  mm,	Z =   -237.136  mm,
	W =  90.000 deg,	P =   0.000 deg,	R =   90.000 deg
};
P[849]{
   GP1:
	UF : 0, UT : 6,		CONFIG : 'N U T, 0, 0, 0',
	X =  261.849  mm,	Y =   -340.709  mm,	Z =   -237.505  mm,
	W =  90.000 deg,	P =   0.000 deg,	R =   90.000 deg
};
P[850]{
   GP1:
	UF : 0, UT : 6,		CONFIG : 'N U T, 0, 0, 0',
	X =  261.482  mm,	Y =   -340.066  mm,	Z =   -237.448  mm,
	W =  90.000 deg,	P =   0.000 deg,	R =   90.000 deg
};
P[851]{
   GP1:
	UF : 0, UT : 6,		CONFIG : 'N U T, 0, 0, 0',
	X =  261.129  mm,	Y =   -339.412  mm,	Z =   -237.138  mm,
	W =  90.000 deg,	P =   0.000 deg,	R =   90.000 deg
};
P[852]{
   GP1:
	UF : 0, UT : 6,		CONFIG : 'N U T, 0, 0, 0',
	X =  260.949  mm,	Y =   -339.154  mm,	Z =   -237.520  mm,
	W =  90.000 deg,	P =   0.000 deg,	R =   90.000 deg
};
P[853]{
   GP1:
	UF : 0, UT : 6,		CONFIG : 'N U T, 0, 0, 0',
	X =  260.485  mm,	Y =   -338.345  mm,	Z =   -237.490  mm,
	W =  90.000 deg,	P =   0.000 deg,	R =   90.000 deg
};
P[854]{
   GP1:
	UF : 0, UT : 6,		CONFIG : 'N U T, 0, 0, 0',
	X =  260.110  mm,	Y =   -337.704  mm,	Z =   -237.549  mm,
	W =  90.000 deg,	P =   0.000 deg,	R =   90.000 deg
};
P[855]{
   GP1:
	UF : 0, UT : 6,		CONFIG : 'N U T, 0, 0, 0',
	X =  259.235  mm,	Y =   -336.129  mm,	Z =   -237.123  mm,
	W =  90.000 deg,	P =   0.000 deg,	R =   90.000 deg
};
P[856]{
   GP1:
	UF : 0, UT : 6,		CONFIG : 'N U T, 0, 0, 0',
	X =  258.490  mm,	Y =   -334.903  mm,	Z =   -237.579  mm,
	W =  90.000 deg,	P =   0.000 deg,	R =   90.000 deg
};
P[857]{
   GP1:
	UF : 0, UT : 6,		CONFIG : 'N U T, 0, 0, 0',
	X =  258.394  mm,	Y =   -334.671  mm,	Z =   -237.114  mm,
	W =  90.000 deg,	P =   0.000 deg,	R =   90.000 deg
};
P[858]{
   GP1:
	UF : 0, UT : 6,		CONFIG : 'N U T, 0, 0, 0',
	X =  257.561  mm,	Y =   -333.272  mm,	Z =   -237.422  mm,
	W =  90.000 deg,	P =   0.000 deg,	R =   90.000 deg
};
P[859]{
   GP1:
	UF : 0, UT : 6,		CONFIG : 'N U T, 0, 0, 0',
	X =  257.141  mm,	Y =   -332.541  mm,	Z =   -237.395  mm,
	W =  90.000 deg,	P =   0.000 deg,	R =   90.000 deg
};
P[860]{
   GP1:
	UF : 0, UT : 6,		CONFIG : 'N U T, 0, 0, 0',
	X =  256.821  mm,	Y =   -331.951  mm,	Z =   -237.131  mm,
	W =  90.000 deg,	P =   0.000 deg,	R =   90.000 deg
};
P[861]{
   GP1:
	UF : 0, UT : 6,		CONFIG : 'N U T, 0, 0, 0',
	X =  256.333  mm,	Y =   -331.150  mm,	Z =   -237.463  mm,
	W =  90.000 deg,	P =   0.000 deg,	R =   90.000 deg
};
P[862]{
   GP1:
	UF : 0, UT : 6,		CONFIG : 'N U T, 0, 0, 0',
	X =  255.846  mm,	Y =   -330.258  mm,	Z =   -237.113  mm,
	W =  90.000 deg,	P =   0.000 deg,	R =   90.000 deg
};
P[863]{
   GP1:
	UF : 0, UT : 6,		CONFIG : 'N U T, 0, 0, 0',
	X =  255.490  mm,	Y =   -329.700  mm,	Z =   -237.530  mm,
	W =  90.000 deg,	P =   0.000 deg,	R =   90.000 deg
};
P[864]{
   GP1:
	UF : 0, UT : 6,		CONFIG : 'N U T, 0, 0, 0',
	X =  255.001  mm,	Y =   -328.856  mm,	Z =   -237.547  mm,
	W =  90.000 deg,	P =   0.000 deg,	R =   90.000 deg
};
P[865]{
   GP1:
	UF : 0, UT : 6,		CONFIG : 'N U T, 0, 0, 0',
	X =  254.597  mm,	Y =   -328.207  mm,	Z =   -237.528  mm,
	W =  90.000 deg,	P =   0.000 deg,	R =   90.000 deg
};
P[866]{
   GP1:
	UF : 0, UT : 6,		CONFIG : 'N U T, 0, 0, 0',
	X =  253.362  mm,	Y =   -326.686  mm,	Z =   -237.548  mm,
	W =  90.000 deg,	P =   0.000 deg,	R =   90.000 deg
};
P[867]{
   GP1:
	UF : 0, UT : 6,		CONFIG : 'N U T, 0, 0, 0',
	X =  252.321  mm,	Y =   -325.794  mm,	Z =   -237.387  mm,
	W =  90.000 deg,	P =   0.000 deg,	R =   90.000 deg
};
P[868]{
   GP1:
	UF : 0, UT : 6,		CONFIG : 'N U T, 0, 0, 0',
	X =  251.205  mm,	Y =   -325.167  mm,	Z =   -237.590  mm,
	W =  90.000 deg,	P =   0.000 deg,	R =   90.000 deg
};
P[869]{
   GP1:
	UF : 0, UT : 6,		CONFIG : 'N U T, 0, 0, 0',
	X =  249.670  mm,	Y =   -324.567  mm,	Z =   -237.319  mm,
	W =  90.000 deg,	P =   0.000 deg,	R =   90.000 deg
};
P[870]{
   GP1:
	UF : 0, UT : 6,		CONFIG : 'N U T, 0, 0, 0',
	X =  242.130  mm,	Y =   -326.038  mm,	Z =   -237.461  mm,
	W =  90.000 deg,	P =   0.000 deg,	R =   90.000 deg
};
P[871]{
   GP1:
	UF : 0, UT : 6,		CONFIG : 'N U T, 0, 0, 0',
	X =  240.646  mm,	Y =   -326.901  mm,	Z =   -237.527  mm,
	W =  90.000 deg,	P =   0.000 deg,	R =   90.000 deg
};
P[872]{
   GP1:
	UF : 0, UT : 6,		CONFIG : 'N U T, 0, 0, 0',
	X =  239.820  mm,	Y =   -327.382  mm,	Z =   -237.589  mm,
	W =  90.000 deg,	P =   0.000 deg,	R =   90.000 deg
};
P[873]{
   GP1:
	UF : 0, UT : 6,		CONFIG : 'N U T, 0, 0, 0',
	X =  239.207  mm,	Y =   -327.730  mm,	Z =   -237.515  mm,
	W =  90.000 deg,	P =   0.000 deg,	R =   90.000 deg
};
P[874]{
   GP1:
	UF : 0, UT : 6,		CONFIG : 'N U T, 0, 0, 0',
	X =  237.669  mm,	Y =   -328.624  mm,	Z =   -237.587  mm,
	W =  90.000 deg,	P =   0.000 deg,	R =   90.000 deg
};
P[875]{
   GP1:
	UF : 0, UT : 6,		CONFIG : 'N U T, 0, 0, 0',
	X =  236.924  mm,	Y =   -329.020  mm,	Z =   -237.157  mm,
	W =  90.000 deg,	P =   0.000 deg,	R =   90.000 deg
};
P[876]{
   GP1:
	UF : 0, UT : 6,		CONFIG : 'N U T, 0, 0, 0',
	X =  235.447  mm,	Y =   -329.905  mm,	Z =   -237.555  mm,
	W =  90.000 deg,	P =   0.000 deg,	R =   90.000 deg
};
P[877]{
   GP1:
	UF : 0, UT : 6,		CONFIG : 'N U T, 0, 0, 0',
	X =  234.683  mm,	Y =   -330.348  mm,	Z =   -237.581  mm,
	W =  90.000 deg,	P =   0.000 deg,	R =   90.000 deg
};
P[878]{
   GP1:
	UF : 0, UT : 6,		CONFIG : 'N U T, 0, 0, 0',
	X =  233.161  mm,	Y =   -331.222  mm,	Z =   -237.523  mm,
	W =  90.000 deg,	P =   0.000 deg,	R =   90.000 deg
};
P[879]{
   GP1:
	UF : 0, UT : 6,		CONFIG : 'N U T, 0, 0, 0',
	X =  231.756  mm,	Y =   -332.002  mm,	Z =   -237.131  mm,
	W =  90.000 deg,	P =   0.000 deg,	R =   90.000 deg
};
P[880]{
   GP1:
	UF : 0, UT : 6,		CONFIG : 'N U T, 0, 0, 0',
	X =  230.225  mm,	Y =   -332.887  mm,	Z =   -237.147  mm,
	W =  90.000 deg,	P =   0.000 deg,	R =   90.000 deg
};
P[881]{
   GP1:
	UF : 0, UT : 6,		CONFIG : 'N U T, 0, 0, 0',
	X =  229.674  mm,	Y =   -333.236  mm,	Z =   -237.533  mm,
	W =  90.000 deg,	P =   0.000 deg,	R =   90.000 deg
};
P[882]{
   GP1:
	UF : 0, UT : 6,		CONFIG : 'N U T, 0, 0, 0',
	X =  226.612  mm,	Y =   -335.009  mm,	Z =   -237.588  mm,
	W =  90.000 deg,	P =   0.000 deg,	R =   90.000 deg
};
P[883]{
   GP1:
	UF : 0, UT : 6,		CONFIG : 'N U T, 0, 0, 0',
	X =  225.879  mm,	Y =   -335.423  mm,	Z =   -237.476  mm,
	W =  90.000 deg,	P =   0.000 deg,	R =   90.000 deg
};
P[884]{
   GP1:
	UF : 0, UT : 6,		CONFIG : 'N U T, 0, 0, 0',
	X =  225.227  mm,	Y =   -335.774  mm,	Z =   -237.156  mm,
	W =  90.000 deg,	P =   0.000 deg,	R =   90.000 deg
};
P[885]{
   GP1:
	UF : 0, UT : 6,		CONFIG : 'N U T, 0, 0, 0',
	X =  224.533  mm,	Y =   -336.171  mm,	Z =   -237.119  mm,
	W =  90.000 deg,	P =   0.000 deg,	R =   90.000 deg
};
P[886]{
   GP1:
	UF : 0, UT : 6,		CONFIG : 'N U T, 0, 0, 0',
	X =  223.736  mm,	Y =   -336.666  mm,	Z =   -237.544  mm,
	W =  90.000 deg,	P =   0.000 deg,	R =   90.000 deg
};
P[887]{
   GP1:
	UF : 0, UT : 6,		CONFIG : 'N U T, 0, 0, 0',
	X =  222.986  mm,	Y =   -337.099  mm,	Z =   -237.542  mm,
	W =  90.000 deg,	P =   0.000 deg,	R =   90.000 deg
};
P[888]{
   GP1:
	UF : 0, UT : 6,		CONFIG : 'N U T, 0, 0, 0',
	X =  221.492  mm,	Y =   -337.962  mm,	Z =   -237.551  mm,
	W =  90.000 deg,	P =   0.000 deg,	R =   90.000 deg
};
P[889]{
   GP1:
	UF : 0, UT : 6,		CONFIG : 'N U T, 0, 0, 0',
	X =  220.794  mm,	Y =   -338.368  mm,	Z =   -237.582  mm,
